ABB RAPID module: ToolPaths.mod

MODULE ToolPaths

    PERS jointtarget CurrentJoints5:=[[111.289,20.3366,35.7518,0.0387684,32.6999,-249.807],[1082.85,9E+09,9E+09,9E+09,9E+09,9E+09]];
    PERS jointtarget CurrentJoints6:=[[105.901,37.7221,15.0236,0.230043,36.0283,-255.346],[1082.85,9E+09,9E+09,9E+09,9E+09,9E+09]];


    TASK PERS wobjdata Bed1:=[FALSE,TRUE,"",[[1000.00,930.569,220.66],[1,0.000655845,-0.000507562,-0.00020191]],[[0,0,0],[1,0,0,0]]];
    !Z 185.66
    !Track -230.02 at measurement

    PERS robtarget pScreed1:=[[-1100,1500,1500],[0.00814298,0.999961,0.000966756,0.00335392],[0,-1,-2,0],[-300,9E+09,9E+09,9E+09,9E+09,9E+09]];
    PERS robtarget pScreed2:=[[-1100,1500,1500],[0.00814298,0.999961,0.000966756,0.00335392],[0,-1,-2,0],[-300,9E+09,9E+09,9E+09,9E+09,9E+09]];

    CONST num HeliOverlapMin:=450;
    CONST num PanOverlapMin:=450;
    CONST num HeliBladeWidth:=1150;
    VAR num HeliPasses;
    VAR num HeliPassWidth;
    CONST num ScreedYpos:=2955;
    CONST num wBedXmin:=1600;
    CONST num wBedXmax:=10200;
    CONST num wBedYmin:=955;
    CONST num wBedYmax:=4955;
    CONST num FormHeight:=150;
    CONST num FormWidth:=65;
    PERS num PitchZOffset:=0;

    VAR speeddata vVS:=[50,15,2000,15];
    ![mm/s TCP, degrees/s TCP, mm/s external axes, degrees/s external axes]
    VAR speeddata vHeli:=[40,10,2000,15];
    VAR speeddata vPlotter:=[1000,30,2000,15];
    VAR zonedata zVS:=z5;
    VAR zonedata zHeli:=z5;
    VAR zonedata zPlotter:=z0;


    VAR robtarget Plotterp1:=[[1000,1000,-10],[0.000337803,0.93262,-0.36086,0.000225436],[0,-1,-2,0],[3400,9E+09,9E+09,9E+09,9E+09,9E+09]];
    PERS robtarget Plotterp2:=[[-2250,790,-20],[6.12303E-17,1,0,0],[0,-1,-1,0],[8453.51,9E+09,9E+09,9E+09,9E+09,9E+09]];
    PERS robtarget Plotterp3:=[[-6000,3500,-20],[4.32964E-17,0.707107,-0.707107,-4.32964E-17],[0,-1,-1,0],[1989.63,9E+09,9E+09,9E+09,9E+09,9E+09]];
    PERS robtarget Plotterp4:=[[-6000,500,-20],[6.12303E-17,1,0,0],[1,-1,0,0],[4703.51,9E+09,9E+09,9E+09,9E+09,9E+09]];
    PERS robtarget Plotterp5:=[[1000,1000,-20],[5.65694E-17,0.92388,-0.382683,-2.34318E-17],[1,-1,0,0],[390.38,9E+09,9E+09,9E+09,9E+09,9E+09]];
    PERS robtarget Plotterc5:=[[-2250,3250,-20],[0.00237199,0.67253,-0.740066,0.000521901],[0,-1,-1,0],[0,9E+09,9E+09,9E+09,9E+09,9E+09]];
    VAR num Plotterc5r:=500;
    VAR robtarget PlotterTemp:=[[1500,3000,-10],[0.00237199,0.67253,-0.740066,0.000521901],[0,-1,-1,0],[3400,9E+09,9E+09,9E+09,9E+09,9E+09]];
    VAR robtarget PlotterTemp2:=[[1500,3000,-10],[0.00237199,0.67253,-0.740066,0.000521901],[0,-1,-1,0],[3400,9E+09,9E+09,9E+09,9E+09,9E+09]];
    VAR robtarget PlotterTemp3:=[[1500,3000,-10],[0.00237199,0.67253,-0.740066,0.000521901],[0,-1,-1,0],[3400,9E+09,9E+09,9E+09,9E+09,9E+09]];
    VAR num PlotterZ:=0;
    VAR num PlotterZOri;

    VAR robtarget pHeliStart:=[[-900,900,163.71],[0.000446787,0.711247,-0.702933,-0.00362622],[1,0,0,0],[7000,9E+09,9E+09,9E+09,9E+09,9E+09]];
    ![0.00497429,-0.71119,0.702786,0.0165738],[0,0,-1,0]
    VAR robtarget pHeliEnd:=[[-2590,2800,163.71],[0.000446787,0.711247,-0.702933,-0.00362622],[1,0,0,0],[5500,9E+09,9E+09,9E+09,9E+09,9E+09]];
    !154.71],[0.000446787,0.711247,-0.702933,-0.00362622],[1,0,0,0]
    VAR robtarget pHeliTempS;
    VAR robtarget pHeliTempE;
    VAR robtarget pHeliTemp1;
    VAR robtarget pHeliTemp2;

    VAR robtarget pScreedStart:=[[500,1900,145],[0.00523034,0.999956,0.00749019,-0.00219287],[0,-1,-2,0],[2000,9E+09,9E+09,9E+09,9E+09,9E+09]];
    VAR robtarget pScreedEnd:=[[6500,1900,145],[0.00523034,0.999956,0.00749019,-0.00219287],[0,-1,-2,0],[7700,9E+09,9E+09,9E+09,9E+09,9E+09]];


    VAR num iTaskno:=-1;
    VAR num iPlotType:=-1;
    VAR num iAngle:=-1;
    VAR num iPlotSide:=-1;
    VAR num iCoord1x:=-1;
    VAR num iCoord1y:=-1;
    VAR num iCoord2x:=-1;
    VAR num iCoord2y:=-1;
    VAR num iCoord3x:=-1;
    VAR num iCoord3y:=-1;
    VAR num iCoord4x:=-1;
    VAR num iCoord4y:=-1;
    VAR num iCoordTemp:=-1;
    VAR num iHeliBladeSpeed:=-1;
    VAR num iHeliBladeAngle:=-1;
    VAR num iZoffset:=0;
    VAR num iHeliPan:=-1;
    VAR num iLRUD:=-1;

    CONST num TieInWidth:=25;
    CONST num GroutWidth:=50;
    CONST num GroutHeight:=500;
    CONST num TriangleBase:=25;
    CONST num TriangleHeight:=50;
    CONST num PlotCircleD:=60;
    VAR num TriangleAngle:=0;
    VAR num CrossHairExt:=10;

    CONST num BedXmin:=10;
    CONST num BedXmax:=8000;
    CONST num BedYmin:=10;
    CONST num BedYmax:=3800;

    CONST num PlotA6Max:=45;
    !45;
    CONST num PlotWaitTime:=0.3;
    PERS num anglex:=179.861;
    PERS num angley:=-0.241379;
    PERS num anglez:=-95.4741;
    VAR pose Object;

    PERS num BedZread:=-8.28;

    VAR robtarget p10maps:=[[-350,150,250],[0.00321343,0.67631,-0.736609,0.000689698],[0,0,-1,0],[7700,9E+09,9E+09,9E+09,9E+09,9E+09]];

    !VAR num BedZreads{4,24}:=[
    !  [13.28, 12.88, 12.68, 14.03, 15.46, 10.94,  8.17,  6.79,  4.83,  2.37,  0.97,  0.30,  0.00,  0.24,  0.47, 0, 0, 0, 0, 0, 0, 0, 0, 0],
    !  [15.76, 14.97, 14.36, 15.69, 16.55, 13.22, 10.94,  9.86,  7.97,  6.00,  4.27,  3.57,  2.82,  2.70,  1.69, 0, 0, 0, 0, 0, 0, 0, 0, 0],
    !  [16.92, 16.33, 16.18, 17.01, 17.20, 14.79, 12.97, 12.12, 10.27,  8.39,  6.92,  5.72,  4.82,  4.65,  2.84, 0, 0, 0, 0, 0, 0, 0, 0, 0],
    !  [17.97, 18.08, 18.34, 18.15, 17.16, 15.42, 14.97, 14.02, 12.65, 11.42,  9.54,  8.23,  6.97,  6.59,  4.58, 0, 0, 0, 0, 0, 0, 0, 0, 0]
    !];

    VAR num BedZreads{4,24}:=[
  [2.28,1.88,1.68,3.03,4.46,-0.06,-2.83,-4.21,-6.17,-8.63,-10.03,-10.70,-11.00,-10.76,-10.53,0,0,0,0,0,0,0,0,0],
  [4.76,3.97,3.36,4.69,5.55,2.22,-0.06,-1.14,-3.03,-5.00,-6.73,-7.43,-8.18,-8.30,-9.31,0,0,0,0,0,0,0,0,0],
  [5.92,5.33,5.18,6.01,6.20,3.79,1.97,1.12,-0.73,-2.61,-4.08,-5.28,-6.18,-6.35,-8.16,0,0,0,0,0,0,0,0,0],
  [6.97,7.08,7.34,7.15,6.16,4.42,3.97,3.02,1.65,0.42,-1.46,-2.77,-4.03,-4.41,-6.42,0,0,0,0,0,0,0,0,0]
];

    VAR num BedZpos{4,24,2}:=[[
    [-350,2100],[-850,2100],[-1350,2100],[-1850,2100],[-2350,2100],[-2850,2100],[-3350,2100],[-3850,2100],[-4350,2100],[-4850,2100],[-5350,2100],[-5850,2100],[-6350,2100],[-6850,2100],[-7350,2100],[-7850,2100],[-8350,2100],[0,0],[0,0],[0,0],[0,0],[0,0],[0,0],[0,0]],

   [[-350,1450],[-850,1450],[-1350,1450],[-1850,1450],[-2350,1450],[-2850,1450],[-3350,1450],[-3850,1450],[-4350,1450],[-4850,1450],[-5350,1450],[-5850,1450],[-6350,1450],[-6850,1450],[-7350,1450],[-7850,1450],[-8350,1450],[0,0],[0,0],[0,0],[0,0],[0,0],[0,0],[0,0]],

   [[-350,800],[-850,800],[-1350,800],[-1850,800],[-2350,800],[-2850,800],[-3350,800],[-3850,800],[-4350,800],[-4850,800],[-5350,800],[-5850,800],[-6350,800],[-6850,800],[-7350,800],[-7850,800],[-8350,800],[0,0],[0,0],[0,0],[0,0],[0,0],[0,0],[0,0]],

    [[-350,150],[-850,150],[-1350,150],[-1850,150],[-2350,150],[-2850,150],[-3350,150],[-3850,150],[-4350,150],[-4850,150],[-5350,150],[-5850,150],[-6350,150],[-6850,150],[-7350,150],[-7850,150],[-8350,150],[0,0],[0,0],[0,0],[0,0],[0,0],[0,0],[0,0]]];


    PERS num Bed1Zread{10,20}:=[[0,0,0,0,0,0,0,0,0,0,0,0,0,0,0,0,0,0,0,0],
                                 [0,0,0,0,0,0,0,0,0,0,0,0,0,0,0,0,0,0,0,0],
                                 [0,0,0,0,0,0,0,0,0,0,0,0,0,0,0,0,0,0,0,0],
                                 [0,0,0,0,0,0,0,0,0,0,0,0,0,0,0,0,0,0,0,0],
                                 [0,0,0,0,0,0,0,0,0,0,0,0,0,0,0,0,0,0,0,0],
                                 [0,0,0,0,0,0,0,0,0,0,0,0,0,0,0,0,0,0,0,0],
                                 [0,0,0,0,0,0,0,0,0,0,0,0,0,0,0,0,0,0,0,0],
                                 [0,0,0,0,0,0,0,0,0,0,0,0,0,0,0,0,0,0,0,0],
                                 [0,0,0,0,0,0,0,0,0,0,0,0,0,0,0,0,0,0,0,0],
                                 [0,0,0,0,0,0,0,0,0,0,0,0,0,0,0,0,0,0,0,0]];

    PERS num Bed1Zpos{10,20,2}:=[[[0,0],[0,0],[0,0],[0,0],[0,0],[0,0],[0,0],[0,0],[0,0],[0,0],[0,0],[0,0],[0,0],[0,0],[0,0],[0,0],[0,0],[0,0],[0,0],[0,0]],

                               [[0,0],[0,0],[0,0],[0,0],[0,0],[0,0],[0,0],[0,0],[0,0],[0,0],[0,0],[0,0],[0,0],[0,0],[0,0],[0,0],[0,0],[0,0],[0,0],[0,0]],

                               [[0,0],[0,0],[0,0],[0,0],[0,0],[0,0],[0,0],[0,0],[0,0],[0,0],[0,0],[0,0],[0,0],[0,0],[0,0],[0,0],[0,0],[0,0],[0,0],[0,0]],

                               [[0,0],[0,0],[0,0],[0,0],[0,0],[0,0],[0,0],[0,0],[0,0],[0,0],[0,0],[0,0],[0,0],[0,0],[0,0],[0,0],[0,0],[0,0],[0,0],[0,0]],

                               [[0,0],[0,0],[0,0],[0,0],[0,0],[0,0],[0,0],[0,0],[0,0],[0,0],[0,0],[0,0],[0,0],[0,0],[0,0],[0,0],[0,0],[0,0],[0,0],[0,0]],

                               [[0,0],[0,0],[0,0],[0,0],[0,0],[0,0],[0,0],[0,0],[0,0],[0,0],[0,0],[0,0],[0,0],[0,0],[0,0],[0,0],[0,0],[0,0],[0,0],[0,0]],

                               [[0,0],[0,0],[0,0],[0,0],[0,0],[0,0],[0,0],[0,0],[0,0],[0,0],[0,0],[0,0],[0,0],[0,0],[0,0],[0,0],[0,0],[0,0],[0,0],[0,0]],

                               [[0,0],[0,0],[0,0],[0,0],[0,0],[0,0],[0,0],[0,0],[0,0],[0,0],[0,0],[0,0],[0,0],[0,0],[0,0],[0,0],[0,0],[0,0],[0,0],[0,0]],

                               [[0,0],[0,0],[0,0],[0,0],[0,0],[0,0],[0,0],[0,0],[0,0],[0,0],[0,0],[0,0],[0,0],[0,0],[0,0],[0,0],[0,0],[0,0],[0,0],[0,0]],

                               [[0,0],[0,0],[0,0],[0,0],[0,0],[0,0],[0,0],[0,0],[0,0],[0,0],[0,0],[0,0],[0,0],[0,0],[0,0],[0,0],[0,0],[0,0],[0,0],[0,0]]];

    CONST num XGridSpacing:=460;
    CONST num YGridSpacing:=400;


    PERS num ScrInitialD:=50;

    PERS num HeliZOffs:=0;
    !Offset based on bed heights

    VAR num SEnddiv:=0;
    VAR num SStartdiv:=0;

    VAR num ScrBedZ;

    PERS num HeliZArray{30}:=[-50,-50,-50,-50,-50,-50,-50,-50,-50,-50,-50,-50,-50,-50,-50,-50,-50,-50,-50,-50,-50,-50,-50,-50,-50,-50,-50,-50,-50,-50];
    VAR bool WithinBlades:=FALSE;
    PERS num HeliZArrayCounter:=1;
    PERS num HeliDiv:=12;
    PERS num PreviousHighest:=-50;

    !CONST robtarget p10:=[[-8200.58,3455.68,-35.54],[0.000477585,0.709995,-0.70418,0.00603077],[1,-1,0,0],[700.099,9E+09,9E+09,9E+09,9E+09,9E+09]];
    CONST robtarget pVacStart:=[[-8200.58,3455.68,-35.54],[0.00615322,-0.709926,0.704246,-0.00239206],[1,-1,0,0],[700,9E+09,9E+09,9E+09,9E+09,9E+09]];
    CONST robtarget pVacStart2:=[[-72.58,1432.35,-35.54],[0.00615322,-0.709926,0.704246,-0.00239206],[1,-1,0,0],[8680,9E+09,9E+09,9E+09,9E+09,9E+09]];
    VAR num iTask:=-1;
    VAR num iPete:=-1;
    VAR num PeteXoffset:=0;
    VAR num PeteYoffset:=0;
    VAR num FormStartX:=7300;
    VAR num FormStartY:=3500;
    VAR num FormXLength:=4750;
    VAR num FormYlength:=1800;
    VAR num CrnrMarkLngth:=300;
    VAR speeddata PanTrvSpd:=[100,30,2000,15];
    VAR num PanBldSpd:=70;
    VAR num PanZOffset:=0;
    VAR num VSZOffset:=0;
    VAR num VSAngleOffset:=0;
    VAR num DummyRun:=0;
    VAR num DummyZOffs:=0;

    PROC PetePanels()
        PeteYoffset:=0;
        PeteXoffset:=0;
        TPErase;
        TPReadNum iTask,"1:Home,2:PackAway,3:Sync,4:Py_28-jan_4:34pm";
        TEST iTask
        CASE 1:
            Home;
        CASE 4:
            FormXLength:=4750;
            FormYlength:=1800;
            TPErase;
            TPWrite "8:Datum,9:PyHeli,10:PyVac,11:PyPolish";
            TPWrite "12:PyVibScreed,13:PyPan";
            TPReadNum iTaskno,"Enter task #:";
            TEST iTaskno
            CASE 1:
                !                TPReadNum iPete,"Enter X  offset (+mm moves closer to the tools)";
                !                IF iPete>(FormStartX-FormXLength-300) OR iPete<0 THEN
                !                    TPWrite "Invalid offset";
                !                    Stop;
                !                    EXIT;
                !                ELSE
                !                    PeteXoffset:=iPete;
                !                ENDIF

                !                TPReadNum iPete,"Enter Y  offset (+mm moves closer to the track)";
                !                IF iPete>(FormStartY-FormYLength-300) OR iPete<0 THEN
                !                    TPWrite "Invalid offset";
                !                    Stop;
                !                    EXIT;
                !                ELSE
                !                    PeteYoffset:=iPete;
                !                ENDIF

                !Formbox
                PlotRect(FormStartX-FormXLength-PeteXoffset-FormWidth),(FormStartY-FormYLength-PeteYoffset-FormWidth),(FormStartX-FormXLength-PeteXoffset-FormWidth),(FormStartY-PeteYoffset+FormWidth),(FormStartX-PeteXoffset+FormWidth),(FormStartY-PeteYoffset+FormWidth),(FormStartX-PeteXoffset+FormWidth),(FormStartY-FormYLength-PeteYoffset-FormWidth);
                CurrentJoints:=CJointT();
                CurrentPos:=CalcRobT(CurrentJoints,tPlotter\WObj:=Bed1Wyong);
                MoveL Offs(CurrentPos,0,0,(1000-CurrentPos.trans.z)),v100,z5,tPlotter\WObj:=Bed1Wyong;

                PlotlineStartLift(FormStartX-FormXLength-PeteXoffset+CrnrMarkLngth),(FormStartY-FormYLength-PeteYoffset),(FormStartX-FormXLength-PeteXoffset),(FormStartY-FormYLength-PeteYoffset);
                PlotLineEndLift(FormStartX-FormXLength-PeteXoffset),(FormStartY-FormYLength-PeteYoffset),(FormStartX-FormXLength-PeteXoffset),(FormStartY-FormYLength-PeteYoffset-CrnrMarkLngth);

                PlotlineStartLift(FormStartX-FormXLength-PeteXoffset),(FormStartY-PeteYoffset-CrnrMarkLngth),(FormStartX-FormXLength-PeteXoffset),(FormStartY-PeteYoffset);
                PlotLineEndLift(FormStartX-FormXLength-PeteXoffset),(FormStartY-PeteYoffset),(FormStartX-FormXLength-PeteXoffset+CrnrMarkLngth),(FormStartY-PeteYoffset);


                !Ferrules
                iCoord1x:=FormStartX-600-PeteXoffset;
                iCoord1y:=FormStartY-1480-PeteYoffset;
                PlotCirc iCoord1x,iCoord1y,(PlotCircleD/2);
                PlotLine(iCoord1x-PlotCircleD/2-CrossHairExt),iCoord1y,(iCoord1x+PlotCircleD/2+CrossHairExt),iCoord1y;
                PlotLine iCoord1x,(iCoord1y-PlotCircleD/2-CrossHairExt),iCoord1x,(iCoord1y+PlotCircleD/2+CrossHairExt);
                !Lifters
                iCoord1x:=FormStartX-FormXLength-PeteXoffset;
                iCoord1y:=FormStartY+620-FormYlength-PeteYoffset;
                TriangleAngle:=0;
                PlotLineStartLift iCoord1x-TriangleBase/2*Sin(TriangleAngle),iCoord1y-TriangleBase/2*Cos(TriangleAngle),iCoord1x+TriangleBase/2*Sin(TriangleAngle),iCoord1y+TriangleBase/2*Cos(TriangleAngle);
                PlotLineNoLift iCoord1x+TriangleBase/2*Sin(TriangleAngle),iCoord1y+TriangleBase/2*Cos(TriangleAngle),iCoord1x+TriangleHeight*Cos(TriangleAngle),iCoord1y-TriangleHeight*Sin(TriangleAngle);
                PlotLineEndLift iCoord1x+TriangleHeight*Cos(TriangleAngle),iCoord1y-TriangleHeight*Sin(TriangleAngle),iCoord1x-TriangleBase/2*Sin(TriangleAngle),iCoord1y-TriangleBase/2*Cos(TriangleAngle);

                iCoord1x:=FormStartX-FormXLength-PeteXoffset;
                iCoord1y:=FormStartY-620-PeteYoffset;
                TriangleAngle:=0;
                PlotLineStartLift iCoord1x-TriangleBase/2*Sin(TriangleAngle),iCoord1y-TriangleBase/2*Cos(TriangleAngle),iCoord1x+TriangleBase/2*Sin(TriangleAngle),iCoord1y+TriangleBase/2*Cos(TriangleAngle);
                PlotLineNoLift iCoord1x+TriangleBase/2*Sin(TriangleAngle),iCoord1y+TriangleBase/2*Cos(TriangleAngle),iCoord1x+TriangleHeight*Cos(TriangleAngle),iCoord1y-TriangleHeight*Sin(TriangleAngle);
                PlotLineEndLift iCoord1x+TriangleHeight*Cos(TriangleAngle),iCoord1y-TriangleHeight*Sin(TriangleAngle),iCoord1x-TriangleBase/2*Sin(TriangleAngle),iCoord1y-TriangleBase/2*Cos(TriangleAngle);

                iCoord1x:=FormStartX+350-FormXLength-PeteXoffset;
                iCoord1y:=FormStartY-PeteYoffset;
                TriangleAngle:=0;
                PlotLineStartLift iCoord1x-TriangleHeight*Sin(TriangleAngle),iCoord1y-TriangleHeight*Cos(TriangleAngle),iCoord1x-TriangleBase/2*Cos(TriangleAngle),iCoord1y+TriangleBase/2*Sin(TriangleAngle);
                PlotLineNoLift iCoord1x-TriangleBase/2*Cos(TriangleAngle),iCoord1y+TriangleBase/2*Sin(TriangleAngle),iCoord1x+TriangleBase/2*Cos(TriangleAngle),iCoord1y-TriangleBase/2*Sin(TriangleAngle);
                PlotLineEndLift iCoord1x+TriangleBase/2*Cos(TriangleAngle),iCoord1y-TriangleBase/2*Sin(TriangleAngle),iCoord1x-TriangleHeight*Sin(TriangleAngle),iCoord1y-TriangleHeight*Cos(TriangleAngle);

                iCoord1x:=FormStartX+2170-FormXLength-PeteXoffset;
                iCoord1y:=FormStartY-PeteYoffset;
                TriangleAngle:=0;
                PlotLineStartLift iCoord1x-TriangleHeight*Sin(TriangleAngle),iCoord1y-TriangleHeight*Cos(TriangleAngle),iCoord1x-TriangleBase/2*Cos(TriangleAngle),iCoord1y+TriangleBase/2*Sin(TriangleAngle);
                PlotLineNoLift iCoord1x-TriangleBase/2*Cos(TriangleAngle),iCoord1y+TriangleBase/2*Sin(TriangleAngle),iCoord1x+TriangleBase/2*Cos(TriangleAngle),iCoord1y-TriangleBase/2*Sin(TriangleAngle);
                PlotLineEndLift iCoord1x+TriangleBase/2*Cos(TriangleAngle),iCoord1y-TriangleBase/2*Sin(TriangleAngle),iCoord1x-TriangleHeight*Sin(TriangleAngle),iCoord1y-TriangleHeight*Cos(TriangleAngle);

                iCoord1x:=FormStartX-2170-PeteXoffset;
                iCoord1y:=FormStartY-PeteYoffset;
                TriangleAngle:=0;
                PlotLineStartLift iCoord1x-TriangleHeight*Sin(TriangleAngle),iCoord1y-TriangleHeight*Cos(TriangleAngle),iCoord1x-TriangleBase/2*Cos(TriangleAngle),iCoord1y+TriangleBase/2*Sin(TriangleAngle);
                PlotLineNoLift iCoord1x-TriangleBase/2*Cos(TriangleAngle),iCoord1y+TriangleBase/2*Sin(TriangleAngle),iCoord1x+TriangleBase/2*Cos(TriangleAngle),iCoord1y-TriangleBase/2*Sin(TriangleAngle);
                PlotLineEndLift iCoord1x+TriangleBase/2*Cos(TriangleAngle),iCoord1y-TriangleBase/2*Sin(TriangleAngle),iCoord1x-TriangleHeight*Sin(TriangleAngle),iCoord1y-TriangleHeight*Cos(TriangleAngle);

                iCoord1x:=FormStartX-350-PeteXoffset;
                iCoord1y:=FormStartY-PeteYoffset;
                TriangleAngle:=0;
                PlotLineStartLift iCoord1x-TriangleHeight*Sin(TriangleAngle),iCoord1y-TriangleHeight*Cos(TriangleAngle),iCoord1x-TriangleBase/2*Cos(TriangleAngle),iCoord1y+TriangleBase/2*Sin(TriangleAngle);
                PlotLineNoLift iCoord1x-TriangleBase/2*Cos(TriangleAngle),iCoord1y+TriangleBase/2*Sin(TriangleAngle),iCoord1x+TriangleBase/2*Cos(TriangleAngle),iCoord1y-TriangleBase/2*Sin(TriangleAngle);
                PlotLineEndLift iCoord1x+TriangleBase/2*Cos(TriangleAngle),iCoord1y-TriangleBase/2*Sin(TriangleAngle),iCoord1x-TriangleHeight*Sin(TriangleAngle),iCoord1y-TriangleHeight*Cos(TriangleAngle);

                PlotlineStartLift(FormStartX-PeteXoffset-CrnrMarkLngth),(FormStartY-PeteYoffset),(FormStartX-PeteXoffset+FormWidth),(FormStartY-PeteYoffset+FormWidth);
                PlotLineEndLift(FormStartX-PeteXoffset+FormWidth),(FormStartY-PeteYoffset+FormWidth),(FormStartX-PeteXoffset+FormWidth),(FormStartY-PeteYoffset+FormWidth-CrnrMarkLngth);

                !Grout tubes
                iCoord1x:=FormStartX-PeteXoffset;
                iCoord1y:=FormStartY-150-PeteYoffset;
                PlotLine iCoord1x,iCoord1y,(iCoord1x-350),iCoord1y;
                PlotCirc(iCoord1x-300),icoord1y,(PlotCircleD/2);

                iCoord1x:=FormStartX-PeteXoffset;
                iCoord1y:=FormStartY+150-FormYlength-PeteYoffset;
                PlotLine iCoord1x,iCoord1y,(iCoord1x-350),iCoord1y;
                PlotCirc(iCoord1x-300),icoord1y,(PlotCircleD/2);

                PlotlineStartLift(FormStartX-PeteXoffset),(FormStartY-FormYLength-PeteYoffset+CrnrMarkLngth),(FormStartX-PeteXoffset),(FormStartY-FormYLength-PeteYoffset);
                PlotLineEndLift(FormStartX-PeteXoffset),(FormStartY-FormYLength-PeteYoffset),(FormStartX-PeteXoffset-CrnrMarkLngth),(FormStartY-FormYLength-PeteYoffset);

                CurrentJoints:=CJointT();
                CurrentPos:=CalcRobT(CurrentJoints,tPlotter\WObj:=Bed1Wyong);
                MoveL Offs(CurrentPos,0,0,(1000-CurrentPos.trans.z)),v100,z5,tPlotter\WObj:=Bed1Wyong;

                Home;
            CASE 2:
                !                TPReadNum iPete,"Enter X  offset (+mm moves closer to the tools)";
                !                IF iPete>(FormStartX-FormXLength-300) OR iPete<0 THEN
                !                    TPWrite "Invalid offset";
                !                    Stop;
                !                    EXIT;
                !                ELSE
                !                    PeteXoffset:=iPete;
                !                ENDIF

                !                TPReadNum iPete,"Enter Y  offset (+mm moves closer to the track)";
                !                IF iPete>(FormStartY-FormYLength-300) OR iPete<0 THEN
                !                    TPWrite "Invalid offset";
                !                    Stop;
                !                    EXIT;
                !                ELSE
                !                    PeteYoffset:=iPete;
                !                ENDIF
                TPReadNum iPete,"Enter angle offset (+deg angles front down)";
                IF iPete>15 OR iPete<-15 THEN
                    TPWrite "Invalid angle offset";
                    Stop;
                    EXIT;
                ELSE
                    VSAngleOffset:=iPete;
                ENDIF

                TPReadNum iPete,"Enter Z offset(+mm{400max} moves higher, -mm pushes down more)";
                IF iPete>400 OR iPete<-50 THEN
                    TPWrite "Invalid Z offset";
                    Stop;
                    EXIT;
                ELSE
                    VSZOffset:=iPete;
                ENDIF

                Screed(FormStartX-FormXLength-PeteXoffset),(FormStartX-PeteXoffset),VSZOffset,VSAngleOffset;
                Home;
            CASE 3:
                Polish;
                Home;
            CASE 4:
                VacuumBed;
                Home;
            CASE 5:

                TPReadNum iPete,"Enter 0 real run, 1 for dummmy run";
                IF iPete<>0 AND iPete<>1 THEN
                    TPWrite "Invalid entry";
                    Stop;
                    EXIT;
                ELSE
                    DummyRun:=iPete;
                ENDIF

                TPReadNum iPete,"Enter Y offset (+mm moves further away from track)";
                IF iPete>FormYLength OR iPete<0 THEN
                    TPWrite "Invalid offset";
                    Stop;
                    EXIT;
                ELSE
                    FCHeliOffs:=iPete;
                    FCHeliStartX:=FormStartX-FormXLength;
                    FCHeliStartY:=FormStartY-FormYlength+FCHeliOffs;
                    FCHeliEndX:=FormStartX;
                ENDIF

                TPReadNum iPete,"Enter Heli travel speed, mm/s(options: 5,10,20,30,40,50,60,80,100,150,200,500)";
                IF iPete=5 OR iPete=10 OR iPete=20 OR iPete=30 OR iPete=40 OR iPete=50 OR iPete=60 OR iPete=80 OR iPete=100 OR iPete=150 OR iPete=200 OR iPete=500 THEN
                    FCHeliSpd.v_tcp:=iPete;
                ELSE
                    TPWrite "Invalid travel speed";
                    Stop;
                    EXIT;
                ENDIF

                IF DummyRun=0 THEN

                    TPReadNum iPete,"Enter Heli blade speed (either 70, 100 or 140 rpm)";
                    FCHeliBldSpd:=iPete;
                    IF iPete=140 THEN
                        FCHeliLD:=HeliLoad140rpm;
                    ELSEIF iPete=100 THEN
                        FCHeliLD:=HeliLoad100rpm;
                    ELSEIF iPete=70 THEN
                        FCHeliLD:=HeliLoad70rpm;
                    ELSE
                        TPWrite "Invalid blade speed";
                        Stop;
                        EXIT;
                    ENDIF

                    TPReadNum iPete,"Enter blade angle (0 to 10 degrees)";
                    IF iPete>10 OR iPete<0 THEN
                        TPWrite "Invalid blade angle";
                        Stop;
                        EXIT;
                    ELSE
                        FCBladeAngle:=iPete;
                    ENDIF

                    TPReadNum iPete,"Enter Force in Newtons (robot will press down with this value, 1300 max)";
                    IF iPete>1300 OR iPete<0 THEN
                        TPWrite "Invalid offset";
                        Stop;
                        EXIT;
                    ELSE
                        FCHeliFrce:=iPete;
                    ENDIF

                    HeliFC FCHeliStartX,FCHeliStartY,FCHeliEndX,FCHeliSpd,FCHeliBldSpd,FCBladeAngle,FCHeliFrce,FCHeliLD;
                ELSEIF DummyRun=1 THEN
                    HeliFCDummy FCHeliStartX,FCHeliStartY,FCHeliEndX,FCHeliSpd;
                ELSE
                    TPWrite "Invalid selection";
                    Stop;
                    EXIT;
                ENDIF

            CASE 6:

                TPReadNum iPete,"Enter Pan travel speed, mm/s(options: 5,10,20,30,40,50,60,80,100,150,200,500)";
                IF iPete=5 OR iPete=10 OR iPete=20 OR iPete=30 OR iPete=40 OR iPete=50 OR iPete=60 OR iPete=80 OR iPete=100 OR iPete=150 OR iPete=200 OR iPete=500 THEN
                    PanTrvSpd.v_tcp:=iPete;
                ELSE
                    TPWrite "Invalid travel speed";
                    Stop;
                    EXIT;
                ENDIF

                TPReadNum iPete,"Enter 0 real run, 1 for dummmy run";
                IF iPete<>0 AND iPete<>1 THEN
                    TPWrite "Invalid entry";
                    Stop;
                    EXIT;
                ELSE
                    DummyRun:=iPete;
                ENDIF

                IF DummyRun=0 THEN

                    TPReadNum iPete,"Pan rotation speed (rpm, 40-140)";
                    IF iPete>140 OR iPete<40 THEN
                        TPWrite "Invalid Heli speed.";
                        Stop;
                        EXIT;
                    ELSE
                        PanBldSpd:=iPete;
                    ENDIF

                    TPReadNum iPete,"Enter Z offset (+mm has heli higher, -mm pushes down more)";
                    IF iPete>400 OR iPete<-50 THEN
                        TPWrite "Invalid offset";
                        Stop;
                        EXIT;
                    ELSE
                        PanZOffset:=iPete;
                    ENDIF

                    HeliPanLR(FormStartX-FormXLength-PeteXoffset),(FormStartY-FormYLength-PeteYoffset),(FormStartX-PeteXoffset),2500,PanTrvSpd,PanBldSpd,PanZOffset;
                ELSE
                    TPWrite "Invalid selection";
                    Stop;
                    EXIT;
                ENDIF


            CASE 7:
                PolishTest;
            CASE 8:
                Datum;
            CASE 9:
                PyHeli;
            CASE 10:
                PyVac;
            CASE 11:
                PyPolish;
            CASE 12:
                PyVibScreed;
            CASE 13:
                PyPan;
            DEFAULT:
                RAISE ERR_INVALID_INPUT;
            ENDTEST

        CASE 2:
            PackAway;
        CASE 3:
            MoveAbsJ [[86.92,9.65,27.89,0.50,50.60,-4.00],[1388.98,9E9,9E9,9E9,9E9,9E9]],v100,fine,tool0;
            Stop;
        DEFAULT:
            RAISE ERR_INVALID_INPUT;
        ENDTEST
    ERROR
        RAISE ;
    ENDPROC


    PROC DemoScreen()
        TPErase;
        TPReadNum iTask,"1: Demo, 2: Production";
        TEST iTask
        CASE 1:
            TPErase;
            TPReadNum iTaskno,"Enter Demo #: 1: Home, 2: Plot 3: Screed, 4: Polish, 5: Vac";
            TEST iTaskno
            CASE 1:
                Home;
            CASE 2:
                RobbiePlot;
            CASE 3:
                Screed 500,6000,0,11;
            CASE 4:
                PolishDemo;
            CASE 5:
                VacuumBed;
            DEFAULT:
                RAISE ERR_INVALID_INPUT;
            ENDTEST

        CASE 2:
            TaskToDo;
        DEFAULT:
            RAISE ERR_INVALID_INPUT;
        ENDTEST
    ERROR
        RAISE ;
    ENDPROC


    PROC TaskToDo()
        TPErase;
        TPReadNum iTaskno,"Enter task #: 1: Home, 2: Loadout 3: Plot, 4: Screed, 5: Heli, 6: Vac, 7: Polish";
        TEST iTaskno
        CASE 1:
            Home;
        CASE 2:
            Home;
            MoveJ pHomeLoadout,v500,z50,tTCMaster;
        CASE 3:
            TPErase;
            TPWrite "Plotting: Enter 1 for formbox, 2 for circle/cross, 3 for grout tube,";
            TPWrite " 4 for square/cross, 5 for triangle.";
            TPReadNum iPlotType,"Enter Selection:";
            TPErase;
            IF iPlotType=1 THEN
                !Form box
                TPWrite "Enter the coordinates for each corner of the formwork.";
                TPReadNum iCoord1x,"Enter first coordinate X value";
                TPReadNum iCoord1y,"Enter first coordinate y value";
                TPReadNum iCoord2x,"Enter second coordinate X value";
                TPReadNum iCoord2y,"Enter second coordinate y value";
                TPReadNum iCoord3x,"Enter third coordinate X value";
                TPReadNum iCoord3y,"Enter third coordinate y value";
                TPReadNum iCoord4x,"Enter fourth coordinate X value";
                TPReadNum iCoord4y,"Enter fourth coordinate y value";
                IF iCoord1x<BedXmin OR iCoord1y<BedYmin OR iCoord2x<BedXmin OR iCoord2y<BedYmin OR iCoord3x<BedXmin OR iCoord3y<BedYmin OR iCoord4x<BedXmin OR iCoord4y<BedYmin OR iCoord1x>BedXmax OR iCoord1y>BedYmax OR iCoord2x>BedXmax OR iCoord2y>BedYmax OR iCoord3x>BedXmax OR iCoord3y>BedYmax OR iCoord4x>BedXmax OR iCoord4y>BedYmax OR (iCoord1x*iCoord1x+iCoord1y*iCoord1y<2560000) OR (iCoord2x*iCoord2x+iCoord2y*iCoord2y<2560000) OR (iCoord3x*iCoord3x+iCoord3y*iCoord3y<2560000) OR (iCoord4x*iCoord4x+iCoord4y*iCoord4y<2560000) THEN
                    RAISE ERR_INVALID_INPUT;
                ENDIF
                PlotRect iCoord1x,iCoord1y,iCoord2x,iCoord2y,iCoord3x,iCoord3y,iCoord4x,iCoord4y;

            ELSEIF iPlotType=2 THEN
                !ferrule - Circle with cross
                TPWrite "Enter the coordinates for the centre position of the ferrule.";
                TPReadNum iCoord1x,"Enter centre coordinate X value";
                TPReadNum iCoord1y,"Enter centre coordinate y value";

                IF (iCoord1x-PlotCircleD)<BedXmin OR (iCoord1y-PlotCircleD)<BedYmin OR (iCoord1x+PlotCircleD)>BedXmax OR (iCoord1y+PlotCircleD)>BedYmax OR ((iCoord1x-PlotCircleD)*(iCoord1x-PlotCircleD)+(iCoord1y-PlotCircleD)*(iCoord1y-PlotCircleD)<2560000) THEN
                    RAISE ERR_INVALID_INPUT;
                ENDIF
                PlotCirc iCoord1x,iCoord1y,(PlotCircleD/2);
                PlotLine(iCoord1x-PlotCircleD/2-CrossHairExt),iCoord1y,(iCoord1x+PlotCircleD/2+CrossHairExt),iCoord1y;
                PlotLine iCoord1x,(iCoord1y-PlotCircleD/2-CrossHairExt),iCoord1x,(iCoord1y+PlotCircleD/2+CrossHairExt);

            ELSEIF iPlotType=3 THEN
                !Grout Rectangle
                TPWrite "Enter the edge coordinate coordinate, followed by the angle.";
                TPReadNum iCoord1x,"Enter centre coordinate X value";
                TPReadNum iCoord1y,"Enter centre coordinate y value";
                TPWrite "0 degrees is perpendicular, -90 degrees is left/CCW, +90 is right/CW.,";
                TPReadNum iAngle,"Enter the angle";
                TPErase;
                TPWrite "Enter the side for the grout tube to be placed.";
                TPWrite " ------3------ ";
                TPWrite " |           | ";
                TPWrite "2|     X     |4";
                TPWrite " |           | ";
                TPWrite " ------1------ ";
                TPWrite "ROBOT/TRACK SIDE";
                TPReadNum iPlotSide,"Enter side:";

                IF iAngle<-90 OR iAngle>90 THEN
                    RAISE ERR_INVALID_INPUT;
                ENDIF

                TEST iPlotSide
                CASE 1:
                    IF iCoord1x-GroutWidth/2*Cos(iAngle)<BedXmin OR iCoord1y+GroutWidth/2*Sin(iAngle)<BedYmin OR iCoord1x-GroutWidth/2*Cos(iAngle)+GroutHeight*Sin(iAngle)<BedXmin OR iCoord1y+GroutHeight*Cos(iAngle)+GroutWidth/2*Sin(iAngle)<BedYmin OR iCoord1x+GroutWidth/2*Cos(iAngle)+GroutHeight*Sin(iAngle)<BedXmin OR iCoord1y+GroutHeight*Cos(iAngle)-GroutWidth/2*Sin(iAngle)<BedYmin OR iCoord1x+GroutWidth/2*Cos(iAngle)<BedXmin OR iCoord1y-GroutWidth/2*Sin(iAngle)<BedYmin OR ((iCoord1x-GroutHeight)*(iCoord1x-GroutWidth)+(iCoord1y-GroutHeight)*(iCoord1y-GroutWidth)<2560000) THEN
                        RAISE ERR_INVALID_INPUT;
                    ENDIF

                    IF iCoord1x-GroutWidth/2*Cos(iAngle)>BedXmax OR iCoord1y+GroutWidth/2*Sin(iAngle)>BedYmax OR iCoord1x-GroutWidth/2*Cos(iAngle)+GroutHeight*Sin(iAngle)>BedXmax OR iCoord1y+GroutHeight*Cos(iAngle)+GroutWidth/2*Sin(iAngle)>BedYmax OR iCoord1x+GroutWidth/2*Cos(iAngle)+GroutHeight*Sin(iAngle)>BedXmax OR iCoord1y+GroutHeight*Cos(iAngle)-GroutWidth/2*Sin(iAngle)>BedYmax OR iCoord1x+GroutWidth/2*Cos(iAngle)>BedXmax OR iCoord1y-GroutWidth/2*Sin(iAngle)>BedYmax THEN
                        RAISE ERR_INVALID_INPUT;
                    ENDIF

                    PlotRect iCoord1x-GroutWidth/2*Cos(iAngle),iCoord1y+GroutWidth/2*Sin(iAngle),iCoord1x-GroutWidth/2*Cos(iAngle)+GroutHeight*Sin(iAngle),iCoord1y+GroutHeight*Cos(iAngle)+GroutWidth/2*Sin(iAngle),iCoord1x+GroutWidth/2*Cos(iAngle)+GroutHeight*Sin(iAngle),iCoord1y+GroutHeight*Cos(iAngle)-GroutWidth/2*Sin(iAngle),iCoord1x+GroutWidth/2*Cos(iAngle),iCoord1y-GroutWidth/2*Sin(iAngle);

                CASE 2:

                    IF iCoord1x-GroutWidth/2*Sin(iAngle)<BedXmin OR iCoord1y-GroutWidth/2*Cos(iAngle)<BedYmin OR iCoord1x+GroutWidth/2*Sin(iAngle)<BedXmin OR iCoord1y+GroutWidth/2*Cos(iAngle)<BedYmin OR iCoord1x+GroutWidth/2*Sin(iAngle)+GroutHeight*Cos(iAngle)<BedXmin OR iCoord1y-GroutHeight*Sin(iAngle)+GroutWidth/2*Cos(iAngle)<BedYmin OR iCoord1x-GroutWidth/2*Sin(iAngle)+GroutHeight*Cos(iAngle)<BedXmin OR iCoord1y-GroutHeight*Sin(iAngle)-GroutWidth/2*Cos(iAngle)<BedYmin OR ((iCoord1x-GroutHeight)*(iCoord1x-GroutWidth)+(iCoord1y-GroutHeight)*(iCoord1y-GroutWidth)<2560000) THEN
                        RAISE ERR_INVALID_INPUT;
                    ENDIF

                    IF iCoord1x-GroutWidth/2*Sin(iAngle)>BedXmax OR iCoord1y-GroutWidth/2*Cos(iAngle)>BedYmax OR iCoord1x+GroutWidth/2*Sin(iAngle)>BedXmax OR iCoord1y+GroutWidth/2*Cos(iAngle)>BedYmax OR iCoord1x+GroutWidth/2*Sin(iAngle)+GroutHeight*Cos(iAngle)>BedXmax OR iCoord1y-GroutHeight*Sin(iAngle)+GroutWidth/2*Cos(iAngle)>BedYmax OR iCoord1x-GroutWidth/2*Sin(iAngle)+GroutHeight*Cos(iAngle)>BedXmax OR iCoord1y-GroutHeight*Sin(iAngle)-GroutWidth/2*Cos(iAngle)>BedYmax THEN
                        RAISE ERR_INVALID_INPUT;
                    ENDIF

                    PlotRect iCoord1x-GroutWidth/2*Sin(iAngle),iCoord1y-GroutWidth/2*Cos(iAngle),iCoord1x+GroutWidth/2*Sin(iAngle),iCoord1y+GroutWidth/2*Cos(iAngle),iCoord1x+GroutWidth/2*Sin(iAngle)+GroutHeight*Cos(iAngle),iCoord1y-GroutHeight*Sin(iAngle)+GroutWidth/2*Cos(iAngle),iCoord1x-GroutWidth/2*Sin(iAngle)+GroutHeight*Cos(iAngle),iCoord1y-GroutHeight*Sin(iAngle)-GroutWidth/2*Cos(iAngle);

                CASE 3:

                    IF iCoord1x-GroutWidth/2*Cos(iAngle)-GroutHeight*Sin(iAngle)<BedXmin OR iCoord1y-GroutHeight*Cos(iAngle)+GroutWidth/2*Sin(iAngle)<BedYmin OR iCoord1x-GroutWidth/2*Cos(iAngle)<BedXmin OR iCoord1y+GroutWidth/2*Sin(iAngle)<BedYmin OR iCoord1x+GroutWidth/2*Cos(iAngle)<BedXmin OR iCoord1y-GroutWidth/2*Sin(iAngle)<BedYmin OR iCoord1x+GroutWidth/2*Cos(iAngle)-GroutHeight*Sin(iAngle)<BedXmin OR iCoord1y-GroutHeight*Cos(iAngle)-GroutWidth/2*Sin(iAngle)<BedYmin OR ((iCoord1x-GroutHeight)*(iCoord1x-GroutWidth)+(iCoord1y-GroutHeight)*(iCoord1y-GroutWidth)<2560000) THEN
                        RAISE ERR_INVALID_INPUT;
                    ENDIF

                    IF iCoord1x-GroutWidth/2*Cos(iAngle)-GroutHeight*Sin(iAngle)>BedXmax OR iCoord1y-GroutHeight*Cos(iAngle)+GroutWidth/2*Sin(iAngle)>BedYmax OR iCoord1x-GroutWidth/2*Cos(iAngle)>BedXmax OR iCoord1y+GroutWidth/2*Sin(iAngle)>BedYmax OR iCoord1x+GroutWidth/2*Cos(iAngle)>BedXmax OR iCoord1y-GroutWidth/2*Sin(iAngle)>BedYmax OR iCoord1x+GroutWidth/2*Cos(iAngle)-GroutHeight*Sin(iAngle)>BedXmax OR iCoord1y-GroutHeight*Cos(iAngle)-GroutWidth/2*Sin(iAngle)>BedYmax THEN
                        RAISE ERR_INVALID_INPUT;
                    ENDIF

                    PlotRect iCoord1x-GroutWidth/2*Cos(iAngle)-GroutHeight*Sin(iAngle),iCoord1y-GroutHeight*Cos(iAngle)+GroutWidth/2*Sin(iAngle),iCoord1x-GroutWidth/2*Cos(iAngle),iCoord1y+GroutWidth/2*Sin(iAngle),iCoord1x+GroutWidth*Cos(iAngle),iCoord1y-GroutWidth/2*Sin(iAngle),iCoord1x+GroutWidth/2*Cos(iAngle)-GroutHeight*Sin(iAngle),iCoord1y-GroutHeight*Cos(iAngle)-GroutWidth/2*Sin(iAngle);


                CASE 4:

                    IF iCoord1x-GroutWidth/2*Sin(iAngle)-GroutHeight*Cos(iAngle)<BedXmin OR iCoord1y+GroutHeight*Sin(iAngle)-GroutWidth/2*Cos(iAngle)<BedYmin OR iCoord1x+GroutWidth/2*Sin(iAngle)-GroutHeight*Cos(iAngle)<BedXmin OR iCoord1y+GroutHeight*Sin(iAngle)+GroutWidth/2*Cos(iAngle)<BedYmin OR iCoord1x+GroutWidth/2*Sin(iAngle)<BedXmin OR iCoord1y+GroutWidth/2*Cos(iAngle)<BedYmin OR iCoord1x-GroutWidth/2*Sin(iAngle)<BedXmin OR iCoord1y-GroutWidth/2*Cos(iAngle)<BedYmin OR ((iCoord1x-GroutHeight)*(iCoord1x-GroutWidth)+(iCoord1y-GroutHeight)*(iCoord1y-GroutWidth)<2560000) THEN
                        RAISE ERR_INVALID_INPUT;
                    ENDIF

                    IF iCoord1x-GroutWidth/2*Sin(iAngle)-GroutHeight*Cos(iAngle)>BedXmax OR iCoord1y+GroutHeight*Sin(iAngle)-GroutWidth/2*Cos(iAngle)>BedYmax OR iCoord1x+GroutWidth/2*Sin(iAngle)-GroutHeight*Cos(iAngle)>BedXmax OR iCoord1y+GroutHeight*Sin(iAngle)+GroutWidth/2*Cos(iAngle)>BedYmax OR iCoord1x+GroutWidth/2*Sin(iAngle)>BedXmax OR iCoord1y+GroutWidth/2*Cos(iAngle)>BedYmax OR iCoord1x-GroutWidth/2*Sin(iAngle)>BedXmax OR iCoord1y-GroutWidth/2*Cos(iAngle)>BedYmax THEN
                        RAISE ERR_INVALID_INPUT;
                    ENDIF

                    PlotRect iCoord1x-GroutWidth/2*Sin(iAngle)-GroutHeight*Cos(iAngle),iCoord1y+GroutHeight*Sin(iAngle)-GroutWidth/2*Cos(iAngle),iCoord1x+GroutWidth/2*Sin(iAngle)-GroutHeight*Cos(iAngle),iCoord1y+GroutHeight*Sin(iAngle)+GroutWidth/2*Cos(iAngle),iCoord1x+GroutWidth/2*Sin(iAngle),iCoord1y+GroutWidth/2*Cos(iAngle),iCoord1x-GroutWidth/2*Sin(iAngle),iCoord1y-GroutWidth/2*Cos(iAngle);
                DEFAULT:
                    RAISE ERR_INVALID_INPUT;

                ENDTEST

            ELSEIF iPlotType=4 THEN
                ! Rectangle with cross
                TPWrite "Enter the centre coordinate";
                TPReadNum iCoord1x,"Enter centre coordinate X value";
                TPReadNum iCoord1y,"Enter centre coordinate y value";

                IF (iCoord1x-TieInWidth/2)<BedXmin OR (iCoord1y-TieInWidth/2)<BedYmin OR (iCoord1x+TieInWidth/2)>BedXmax OR (iCoord1y+TieInWidth/2)>BedYmax OR (iCoord1x*iCoord1x+iCoord1y*iCoord1y<2560000) THEN
                    RAISE ERR_INVALID_INPUT;
                ENDIF
                PlotRect iCoord1x-TieInWidth/2,iCoord1y-TieInWidth/2,iCoord1x-TieInWidth/2,iCoord1y+TieInWidth/2,iCoord1x+TieInWidth/2,iCoord1y+TieInWidth/2,iCoord1x+TieInWidth/2,iCoord1y-TieInWidth/2;
                PlotLine iCoord1x,iCoord1y-TieInWidth/2,iCoord1x,iCoord1y+TieInWidth/2;
                PlotLine iCoord1x-TieInWidth/2,iCoord1y,iCoord1x+TieInWidth/2,iCoord1y;


            ELSEIF iPlotType=5 THEN
                !triangle
                TPWrite "Enter the edge coordinate and angle";
                TPReadNum iCoord1x,"Enter centre coordinate X value";
                TPReadNum iCoord1y,"Enter centre coordinate y value";
                TPWrite "0 degrees is up, 90 is pointing right/CW, 180 pointing down, 270 pointing left.";
                TPReadNum iAngle,"Enter the angle";

                IF (iAngle>=0 AND iAngle<=45) OR (iAngle>315 AND iAngle<=360) THEN
                    TriangleAngle:=iAngle;
                    IF iCoord1x-TriangleBase/2*Cos(TriangleAngle)<BedXmin OR iCoord1y+TriangleBase/2*Sin(TriangleAngle)<BedYmin OR iCoord1x+TriangleHeight*Sin(TriangleAngle)<BedXmin OR iCoord1y+TriangleHeight*Cos(TriangleAngle)<BedYmin OR iCoord1x+TriangleBase/2*Cos(TriangleAngle)<BedXmin OR iCoord1y-TriangleBase/2*Sin(TriangleAngle)<BedYmin OR iCoord1x-TriangleBase/2*Cos(TriangleAngle)>BedXmax OR iCoord1y+TriangleBase/2*Sin(TriangleAngle)>BedYmax OR iCoord1x+TriangleHeight*Sin(TriangleAngle)>BedXmax OR iCoord1y+TriangleHeight*Cos(TriangleAngle)>BedYmax OR iCoord1x+TriangleBase/2*Cos(TriangleAngle)>BedXmax OR iCoord1y-TriangleBase/2*Sin(TriangleAngle)>BedYmax OR (iCoord1x*iCoord1x+iCoord1y*iCoord1y<2560000) THEN
                        RAISE ERR_INVALID_INPUT;
                    ENDIF
                    PlotLine iCoord1x-TriangleBase/2*Cos(TriangleAngle),iCoord1y+TriangleBase/2*Sin(TriangleAngle),iCoord1x+TriangleHeight*Sin(TriangleAngle),iCoord1y+TriangleHeight*Cos(TriangleAngle);
                    PlotLine iCoord1x+TriangleHeight*Sin(TriangleAngle),iCoord1y+TriangleHeight*Cos(TriangleAngle),iCoord1x+TriangleBase/2*Cos(TriangleAngle),iCoord1y-TriangleBase/2*Sin(TriangleAngle);
                    PlotLine iCoord1x+TriangleBase/2*Cos(TriangleAngle),iCoord1y-TriangleBase/2*Sin(TriangleAngle),iCoord1x-TriangleBase/2*Cos(TriangleAngle),iCoord1y+TriangleBase/2*Sin(TriangleAngle);

                ELSEIF iAngle<=135 AND iAngle>45 THEN
                    TriangleAngle:=iAngle-90;
                    IF iCoord1x-TriangleBase/2*Sin(TriangleAngle)<BedXmin OR iCoord1y-TriangleBase/2*Cos(TriangleAngle)<BedYmin OR iCoord1x+TriangleBase/2*Sin(TriangleAngle)<BedXmin OR iCoord1y-TriangleBase/2*Sin(TriangleAngle)<BedYmin OR iCoord1x+TriangleHeight*Cos(TriangleAngle)<BedXmin OR iCoord1y-TriangleHeight*Sin(TriangleAngle)<BedYmin OR iCoord1x-TriangleBase/2*Sin(TriangleAngle)>BedXmax OR iCoord1y-TriangleBase/2*Cos(TriangleAngle)>BedYmax OR iCoord1x+TriangleBase/2*Sin(TriangleAngle)>BedXmax OR iCoord1y-TriangleBase/2*Sin(TriangleAngle)>BedYmax OR iCoord1x+TriangleHeight*Cos(TriangleAngle)>BedXmax OR iCoord1y-TriangleHeight*Sin(TriangleAngle)>BedYmax OR (iCoord1x*iCoord1x+iCoord1y*iCoord1y<2560000) THEN

                        RAISE ERR_INVALID_INPUT;
                    ENDIF
                    PlotLine iCoord1x-TriangleBase/2*Sin(TriangleAngle),iCoord1y-TriangleBase/2*Cos(TriangleAngle),iCoord1x+TriangleBase/2*Sin(TriangleAngle),iCoord1y+TriangleBase/2*Cos(TriangleAngle);
                    PlotLine iCoord1x+TriangleBase/2*Sin(TriangleAngle),iCoord1y+TriangleBase/2*Cos(TriangleAngle),iCoord1x+TriangleHeight*Cos(TriangleAngle),iCoord1y-TriangleHeight*Sin(TriangleAngle);
                    PlotLine iCoord1x+TriangleHeight*Cos(TriangleAngle),iCoord1y-TriangleHeight*Sin(TriangleAngle),iCoord1x-TriangleBase/2*Sin(TriangleAngle),iCoord1y-TriangleBase/2*Cos(TriangleAngle);

                ELSEIF iAngle<=225 AND iAngle>135 THEN
                    TriangleAngle:=iAngle-180;
                    IF iCoord1x-TriangleHeight*Sin(TriangleAngle)<BedXmin OR iCoord1y-TriangleHeight*Sin(TriangleAngle)<BedYmin OR iCoord1x-TriangleBase/2*Cos(TriangleAngle)<BedXmin OR iCoord1y+TriangleBase/2*Sin(TriangleAngle)<BedYmin OR iCoord1x+TriangleBase/2*Cos(TriangleAngle)<BedXmin OR iCoord1y-TriangleBase/2*Sin(TriangleAngle)<BedYmin OR iCoord1x-TriangleHeight*Sin(TriangleAngle)>BedXmax OR iCoord1y-TriangleHeight*Sin(TriangleAngle)>BedYmax OR iCoord1x-TriangleBase/2*Cos(TriangleAngle)>BedXmax OR iCoord1y+TriangleBase/2*Sin(TriangleAngle)>BedYmax OR iCoord1x+TriangleBase/2*Cos(TriangleAngle)>BedXmax OR iCoord1y-TriangleBase/2*Sin(TriangleAngle)>BedYmax OR (iCoord1x*iCoord1x+iCoord1y*iCoord1y<2560000) THEN

                        RAISE ERR_INVALID_INPUT;
                    ENDIF
                    PlotLine iCoord1x-TriangleHeight*Sin(TriangleAngle),iCoord1y-TriangleHeight*Cos(TriangleAngle),iCoord1x-TriangleBase/2*Cos(TriangleAngle),iCoord1y+TriangleBase/2*Sin(TriangleAngle);
                    PlotLine iCoord1x-TriangleBase/2*Cos(TriangleAngle),iCoord1y+TriangleBase/2*Sin(TriangleAngle),iCoord1x+TriangleBase/2*Cos(TriangleAngle),iCoord1y-TriangleBase/2*Sin(TriangleAngle);
                    PlotLine iCoord1x+TriangleBase/2*Cos(TriangleAngle),iCoord1y-TriangleBase/2*Sin(TriangleAngle),iCoord1x-TriangleHeight*Sin(TriangleAngle),iCoord1y-TriangleHeight*Cos(TriangleAngle);

                ELSEIF iAngle<=315 AND iAngle>225 THEN
                    TriangleAngle:=iAngle-270;
                    IF iCoord1x-TriangleBase/2*Sin(TriangleAngle)<BedXmin OR iCoord1y-TriangleBase/2*Cos(TriangleAngle)<BedYmin OR iCoord1x+TriangleHeight*Cos(TriangleAngle)<BedXmin OR iCoord1y-TriangleHeight*Sin(TriangleAngle)<BedYmin OR iCoord1x+TriangleBase/2*Sin(TriangleAngle)<BedXmin OR iCoord1y+TriangleBase/2*Cos(TriangleAngle)<BedYmin OR iCoord1x-TriangleBase/2*Sin(TriangleAngle)>BedXmax OR iCoord1y-TriangleBase/2*Cos(TriangleAngle)>BedYmax OR iCoord1x+TriangleHeight*Cos(TriangleAngle)>BedXmax OR iCoord1y-TriangleHeight*Sin(TriangleAngle)>BedYmax OR iCoord1x+TriangleBase/2*Sin(TriangleAngle)>BedXmax OR iCoord1y+TriangleBase/2*Cos(TriangleAngle)>BedYmax OR (iCoord1x*iCoord1x+iCoord1y*iCoord1y<2560000) THEN
                        RAISE ERR_INVALID_INPUT;
                    ENDIF

                    PlotLine iCoord1x-TriangleBase/2*Sin(TriangleAngle),iCoord1y-TriangleBase/2*Cos(TriangleAngle),iCoord1x-TriangleHeight*Cos(TriangleAngle),iCoord1y+TriangleHeight*Sin(TriangleAngle);
                    PlotLine iCoord1x-TriangleHeight*Cos(TriangleAngle),iCoord1y+TriangleHeight*Sin(TriangleAngle),iCoord1x+TriangleBase/2*Sin(TriangleAngle),iCoord1y+TriangleBase/2*Cos(TriangleAngle);
                    PlotLine iCoord1x+TriangleBase/2*Sin(TriangleAngle),iCoord1y+TriangleBase/2*Cos(TriangleAngle),iCoord1x-TriangleBase/2*Sin(TriangleAngle),iCoord1y-TriangleBase/2*Cos(TriangleAngle);



                ELSE
                    RAISE ERR_INVALID_INPUT;
                ENDIF

            ELSE
                RAISE ERR_INVALID_INPUT;
            ENDIF

        CASE 4:
            TPWrite "Enter the x coordinates for the start and end positions of the formwork.";
            TPReadNum iCoord1x,"Enter first coordinate X value";
            TPReadNum iCoord2x,"Enter second coordinate x value";
            TPReadNum iZoffset,"Enter Z offset (-ve for lower, +ve for higher, 0 for no change:";
            IF iCoord1x<0 OR iCoord2x<0 OR iCoord1x>7900 OR iCoord2x>7900 THEN
                RAISE ERR_INVALID_INPUT;
            ENDIF

            IF iCoord1x>iCoord2x THEN
                iCoordTemp:=iCoord1x;
                iCoord1x:=iCoord2x;
                iCoord2x:=iCoordTemp;
            ENDIF

            Screed iCoord1x,iCoord2x,iZoffset,11;

        CASE 5:
            TPWrite "Enter the coordinates for the corner closest to the robot home position.";
            TPReadNum iCoord1x,"Enter first coordinate X value";
            TPReadNum iCoord1y,"Enter first coordinate y value";
            TPWrite "Enter the coordinates for the corner furthest from the robot home position.";
            TPReadNum iCoord2x,"Enter second coordinate X value";
            TPReadNum iCoord2y,"Enter second coordinate y value";
            TPReadNum iHeliBladeSpeed,"Enter speed of heli blades (rpm from 0 - 140).";
            TPReadNum iHeliBladeAngle,"Enter heli blade angle (degrees from 0 - 12).";
            TPReadNum iZoffset,"Enter Z offset (-ve for lower, +ve for higher, 0 for no change:";
            TPReadNum iHeliPan,"Enter 1 for pan attachment or 2 for just blades:";
            !TPReadNum iLRUD,"Enter 1 for left/right movement or 2 for up/down movement:";

            IF iCoord1x<0 OR iCoord1y<0 OR iCoord2x<0 OR iCoord2y<0 OR iCoord1x>8800 OR iCoord1y>2400 OR iCoord2x>8800 OR iCoord2y>2400 OR iHeliBladeSpeed<0 OR iHeliBladeSpeed>140 OR iHeliBladeAngle<0 OR iHeliBladeAngle>12 OR iCoord2y<iCoord1y OR iCoord2x<iCoord1x OR iHeliPan<1 OR iHeliPan>2 THEN
                RAISE ERR_INVALID_INPUT;
            ENDIF
            !IF iLRUD=1 THEN
            HeliTrowelLR iCoord1x,iCoord1y,iCoord2x,iCoord2y,iHeliBladeSpeed,iHeliBladeAngle,iZoffset,iHeliPan;
            !ELSEIF iLRUD=2 THEN
            !    HeliTrowelUD iCoord1x,iCoord1y,iCoord2x,iCoord2y,iHeliBladeSpeed,iHeliBladeAngle,iZoffset,iHeliPan;
            !ELSE
            !    RAISE ERR_INVALID_INPUT;
            !ENDIF

        CASE 6:
            VacuumBed;

        CASE 7:
            Polish;
        DEFAULT:
            RAISE ERR_INVALID_INPUT;
        ENDTEST
    ERROR
        RAISE ;
    ENDPROC

    PROC HeliTrowelLR(num HeliStartX,num HeliStartY,num HeliEndX,num HeliEndY,num HeliSpeed,num HeliAngle,num HeliZoffset,num IsPan)

        pHeliStart.trans:=[HeliStartX,HeliStartY,(FormHeight+HeliZoffset)];
        pHeliEnd.trans:=[HeliEndX,HeliEndY,(FormHeight+HeliZoffset)];

        IF ToolNum<>2 THEN
            Home;
            Heli_Pickup;
        ENDIF

        IF pHeliStart.trans.y<1800 THEN
            pHeliStart.extax.eax_a:=Bed1Wyong.uframe.trans.x-pHeliStart.trans.x+1000+HeliBladeWidth/2;
            pHeliEnd.extax.eax_a:=Bed1Wyong.uframe.trans.x-pHeliEnd.trans.x+1000-HeliBladeWidth/2;
        ELSE
            pHeliStart.extax.eax_a:=Bed1Wyong.uframe.trans.x-pHeliStart.trans.x+HeliBladeWidth/2;
            pHeliEnd.extax.eax_a:=Bed1Wyong.uframe.trans.x-pHeliEnd.trans.x-HeliBladeWidth/2;
        ENDIF

        IF (pHeliEnd.trans.y-pHeliStart.trans.y)<HeliBladeWidth THEN
            HeliPasses:=1;
            HeliPassWidth:=0;
        ELSE
            HeliPasses:=((pHeliEnd.trans.y-pHeliStart.trans.y-HeliBladeWidth) DIV HeliOverlapMin);
            IF HeliPasses MOD 2<>0 THEN
                Incr HeliPasses;
            ENDIF
            IF HeliPasses<1 THEN
                HeliPasses:=1;
            ENDIF
            HeliPassWidth:=(pHeliEnd.trans.y-(HeliBladeWidth/2)-(pHeliStart.trans.y+(HeliBladeWidth/2)))/HeliPasses;
        ENDIF

        pHeliTempS:=pHeliStart;
        pHeliTempE:=pHeliEnd;
        pHeliTempS.trans.x:=pHeliStart.trans.x-(HeliBladeWidth/2)+300;
        pHeliTempS.trans.y:=pHeliStart.trans.y+(HeliBladeWidth/2);
        pHeliTempE.trans.x:=pHeliEnd.trans.x-(HeliBladeWidth/2)-300;
        pHeliTempE.trans.y:=pHeliEnd.trans.y-(HeliBladeWidth/2);
        pHeliTempS.trans.z:=FormHeight+HeliZoffset;
        pHeliTempE.trans.z:=FormHeight+HeliZoffset;

        MoveJ Offs(pHeliTempS,0,0,300),v500,z5,tHeli\WObj:=Bed1Wyong;

        IF IsPan=2 THEN
            HeliBlade_Angle HeliAngle;
            HeliBladeSpeed HeliSpeed,"FWD";
            WaitTime\inpos,4;
        ENDIF

        IF IsPan=1 THEN
            MoveJ Offs(pHeliTempS,0,0,75),v500,z5,tHeli\WObj:=Bed1Wyong;
            Stop;
        ENDIF
        HeliZ pHeliTempS.trans.x,pHeliTempS.trans.y,TRUE;
        HeliZOffs:=HighestArray(HeliZArrayCounter);

        MoveL Offs(pHeliTempS,0,0,PitchZOffset+HeliZOffs),v50,z5,tHeli\WObj:=Bed1Wyong;
        pHeliTemp1:=pHeliTempS;
        pHeliTemp2:=pHeliTempS;
        pHeliTemp2.trans.x:=pHeliTempE.trans.x;
        pHeliTemp2.extax.eax_a:=pHeliTempE.extax.eax_a;

        IF IsPan=1 THEN
            Stop;
            HeliBlade_Angle HeliAngle;
            HeliBladeSpeed HeliSpeed,"FWD";
            WaitTime\inpos,5;
        ENDIF

        HeliDiv:=(pHeliTempE.trans.x-pHeliTempS.trans.x) DIV XGridSpacing;

        FOR i FROM 0 to (2*HeliPasses) DO
            IF (i MOD 2)=0 THEN

                !Needs fixing of -1*x
                FOR M FROM 0 TO (HeliDiv-1) DO
                    HeliZ(pHeliTemp1.trans.x-M*XGridSpacing+XGridSpacing),(pHeliTemp1.trans.y+HeliPassWidth*i/2),TRUE;
                    HeliZOffs:=HighestArray(HeliZArrayCounter);
                    IF (HeliPassWidth*i/2+pHeliTemp1.trans.y)>1600 THEN
                        pHeliTemp1.extax.eax_a:=pHeliTemp1.trans.x+Bed1Wyong.uframe.trans.x-M*XGridSpacing;
                    ELSE
                        pHeliTemp1.extax.eax_a:=pHeliTemp1.trans.x+Bed1Wyong.uframe.trans.x+1000-M*XGridSpacing;
                    ENDIF
                    MoveL Offs(pHeliTemp1,-1*M*XGridSpacing,HeliPassWidth*i/2,PitchZOffset+HeliZOffs),vHeli,z5,tHeli\WObj:=Bed1Wyong;
                    !Across Right
                ENDFOR

                IF (HeliPassWidth*i/2+pHeliTemp2.trans.y)>1600 THEN
                    pHeliTemp2.extax.eax_a:=pHeliTemp2.trans.x+Bed1Wyong.uframe.trans.x;
                ELSE
                    pHeliTemp2.extax.eax_a:=pHeliTemp2.trans.x+Bed1Wyong.uframe.trans.x+1000;
                ENDIF
                HeliZ(pHeliTemp2.trans.x),(pHeliTemp1.trans.y+HeliPassWidth*i/2),TRUE;
                HeliZOffs:=HighestArray(HeliZArrayCounter);
                MoveL Offs(pHeliTemp2,0,HeliPassWidth*i/2,PitchZOffset+HeliZOffs),vHeli,z5,tHeli\WObj:=Bed1Wyong;
                !Across Right

                IF i=(2*HeliPasses) THEN
                ELSE
                    HeliZ(pHeliTemp2.trans.x),(pHeliTemp1.trans.y+HeliPassWidth*(i+1)/2),TRUE;
                    HeliZOffs:=HighestArray(HeliZArrayCounter);
                    IF (HeliPassWidth*(i+1)/2+pHeliTemp2.trans.y)>1600 THEN
                        pHeliTemp2.extax.eax_a:=pHeliTemp2.trans.x+Bed1Wyong.uframe.trans.x;
                    ELSE
                        pHeliTemp2.extax.eax_a:=pHeliTemp2.trans.x+Bed1Wyong.uframe.trans.x+1000;
                    ENDIF
                    MoveL Offs(pHeliTemp2,0,HeliPassWidth*(i+1)/2,PitchZOffset+HeliZOffs),vHeli,z5,tHeli\WObj:=Bed1Wyong;
                    !Up

                    FOR M FROM (HeliDiv-1) TO 0 DO
                        HeliZ(pHeliTemp1.trans.x-M*XGridSpacing),(pHeliTemp1.trans.y+HeliPassWidth*(i+1)/2),TRUE;
                        HeliZOffs:=HighestArray(HeliZArrayCounter);
                        IF (HeliPassWidth*(i+1)/2+pHeliTemp1.trans.y)>1600 THEN
                            pHeliTemp1.extax.eax_a:=pHeliTemp1.trans.x+Bed1Wyong.uframe.trans.x-M*XGridSpacing;
                        ELSE
                            pHeliTemp1.extax.eax_a:=pHeliTemp1.trans.x+Bed1Wyong.uframe.trans.x+1000-M*XGridSpacing;
                        ENDIF
                        MoveL Offs(pHeliTemp1,-1*M*XGridSpacing,HeliPassWidth*(i+1)/2,PitchZOffset+HeliZOffs),vHeli,z5,tHeli\WObj:=Bed1Wyong;
                        !Across Left
                    ENDFOR

                ENDIF

            ENDIF
        ENDFOR

        IF IsPan=1 THEN
            WaitTime\InPos,0.1;
            HeliBladeSpeed 0,"FWD";
            WaitTime\inpos,8;
            MoveL Offs(pHeliTemp2,0,HeliPassWidth*2*HeliPasses/2,18+PitchZOffset+HeliZOffs),v50,fine,tHeli\WObj:=Bed1Wyong;
            HeliBladeSpeed 20,"REV";
            WaitTime\inpos,0.6;
            HeliBladeSpeed 0,"FWD";
            Stop;
        ENDIF
        MoveL Offs(pHeliTemp2,0,HeliPassWidth*2*HeliPasses/2,50+PitchZOffset+HeliZOffs),v50,z5,tHeli\WObj:=Bed1Wyong;

        HeliBladeSpeed 0,"FWD";
        CurrentJoints:=CJointT();
        CurrentPos:=CalcRobT(CurrentJoints,tHeli\WObj:=wobj0);
        MoveJ Offs(pHeliTemp2,0,2500-CurrentPos.trans.y,300),v500,z5,tHeli\WObj:=Bed1Wyong;
        MoveJ Offs(ptHeli,0,0,500),v500,fine,tHeli;

    ENDPROC

    PROC HeliPanLR(num HeliStartX,num HeliStartY,num HeliEndX,num HeliEndY,speeddata HeliVTCP,num HeliSpeed,num HeliZoffset)

        pHeliStart.trans:=[-1*HeliStartX,HeliStartY,(FormHeight+14+HeliZoffset)];
        pHeliEnd.trans:=[-1*HeliEndX,HeliEndY,(FormHeight+14+HeliZoffset)];

        IF ToolNum<>2 THEN
            Home;
            Heli_Pickup;
        ELSE
            pTemp:=ptHeli;
            pTemp.extax.eax_a:=ptHeli.extax.eax_a-2000;
            pTemp.trans.z:=ptHeli.trans.z+800;
            MoveJ Offs(pTemp,-2000,0,0),v500,fine,tHeli;
        ENDIF

        IF pHeliStart.trans.y<1800 THEN
            pHeliStart.extax.eax_a:=Bed1Wyong.uframe.trans.x+pHeliStart.trans.x+1000+HeliBladeWidth/2;
            pHeliEnd.extax.eax_a:=Bed1Wyong.uframe.trans.x+pHeliEnd.trans.x+1000-HeliBladeWidth/2;
        ELSE
            pHeliStart.extax.eax_a:=Bed1Wyong.uframe.trans.x+pHeliStart.trans.x+HeliBladeWidth/2;
            pHeliEnd.extax.eax_a:=Bed1Wyong.uframe.trans.x+pHeliEnd.trans.x-HeliBladeWidth/2;
        ENDIF

        IF (pHeliEnd.trans.y-pHeliStart.trans.y)<HeliBladeWidth THEN
            HeliPasses:=1;
            HeliPassWidth:=0;
        ELSE
            HeliPasses:=((pHeliEnd.trans.y-pHeliStart.trans.y-HeliBladeWidth) DIV PanOverlapMin);
            IF HeliPasses MOD 2<>0 THEN
                Incr HeliPasses;
            ENDIF
            IF HeliPasses<1 THEN
                HeliPasses:=1;
            ENDIF
            HeliPassWidth:=(pHeliEnd.trans.y-(HeliBladeWidth/2)-(pHeliStart.trans.y+(HeliBladeWidth/2)))/HeliPasses;
        ENDIF

        pHeliTempS:=pHeliStart;
        pHeliTempE:=pHeliEnd;
        pHeliTempS.trans.x:=pHeliStart.trans.x+(HeliBladeWidth/2)-300;
        pHeliTempS.trans.y:=pHeliStart.trans.y+(HeliBladeWidth/2);
        pHeliTempE.trans.x:=pHeliEnd.trans.x-(HeliBladeWidth/2)+300;
        pHeliTempE.trans.y:=pHeliEnd.trans.y-(HeliBladeWidth/2);
        pHeliTempS.trans.z:=FormHeight+HeliZoffset;
        pHeliTempE.trans.z:=FormHeight+HeliZoffset;

        MoveJ Offs(pHeliTempS,0,0,300),v500,z5,tHeli\WObj:=Bed1Wyong;

        MoveJ Offs(pHeliTempS,0,0,75),v500,z5,tHeli\WObj:=Bed1Wyong;
        TPWrite "Place pan under blades.";
        Stop;

        HeliZ pHeliTempS.trans.x,pHeliTempS.trans.y,TRUE;
        HeliZOffs:=HighestArray(HeliZArrayCounter);

        MoveL Offs(pHeliTempS,0,0,PitchZOffset+HeliZOffs),v50,z5,tHeli\WObj:=Bed1Wyong;
        pHeliTemp1:=pHeliTempS;
        pHeliTemp2:=pHeliTempS;
        pHeliTemp2.trans.x:=pHeliTempE.trans.x;
        pHeliTemp2.extax.eax_a:=pHeliTempE.extax.eax_a;

        TPWrite "Check blades are under tabs plane";
        Stop;
        HeliBlade_Angle 0;
        HeliBladeSpeed HeliSpeed,"FWD";
        WaitTime\inpos,5;

        HeliDiv:=(abs(pHeliTempE.trans.x)-abs(pHeliTempS.trans.x)) DIV XGridSpacing;

        FOR i FROM 0 to (2*HeliPasses) DO
            IF (i MOD 2)=0 THEN


                FOR M FROM 0 TO (HeliDiv-1) DO
                    HeliZ(pHeliTemp1.trans.x-M*XGridSpacing-XGridSpacing),(pHeliTemp1.trans.y+HeliPassWidth*i/2),TRUE;
                    HeliZOffs:=HighestArray(HeliZArrayCounter);
                    IF (HeliPassWidth*i/2+pHeliTemp1.trans.y)>1600 THEN
                        pHeliTemp1.extax.eax_a:=Bed1Wyong.uframe.trans.x+pHeliTemp1.trans.x-M*XGridSpacing;
                    ELSE
                        pHeliTemp1.extax.eax_a:=Bed1Wyong.uframe.trans.x+pHeliTemp1.trans.x+1000-M*XGridSpacing;
                    ENDIF
                    MoveL Offs(pHeliTemp1,-1*M*XGridSpacing,HeliPassWidth*i/2,PitchZOffset+HeliZOffs),HeliVTCP,z5,tHeli\WObj:=Bed1Wyong;
                    !Across Left
                ENDFOR

                IF (HeliPassWidth*i/2+pHeliTemp2.trans.y)>1600 THEN
                    pHeliTemp2.extax.eax_a:=Bed1Wyong.uframe.trans.x+pHeliTemp2.trans.x;
                ELSE
                    pHeliTemp2.extax.eax_a:=Bed1Wyong.uframe.trans.x+pHeliTemp2.trans.x+1000;
                ENDIF
                HeliZ(pHeliTemp2.trans.x),(pHeliTemp1.trans.y+HeliPassWidth*i/2),TRUE;
                HeliZOffs:=HighestArray(HeliZArrayCounter);
                MoveL Offs(pHeliTemp2,0,HeliPassWidth*i/2,PitchZOffset+HeliZOffs),HeliVTCP,z5,tHeli\WObj:=Bed1Wyong;
                !Across Left final position

                IF i=(2*HeliPasses) THEN
                ELSE
                    HeliZ(pHeliTemp2.trans.x),(pHeliTemp1.trans.y+HeliPassWidth*(i+1)/2),TRUE;
                    HeliZOffs:=HighestArray(HeliZArrayCounter);
                    IF (HeliPassWidth*(i+1)/2+pHeliTemp2.trans.y)>1600 THEN
                        pHeliTemp2.extax.eax_a:=Bed1Wyong.uframe.trans.x+pHeliTemp2.trans.x;
                    ELSE
                        pHeliTemp2.extax.eax_a:=Bed1Wyong.uframe.trans.x+pHeliTemp2.trans.x+1000;
                    ENDIF
                    MoveL Offs(pHeliTemp2,0,HeliPassWidth*(i+1)/2,PitchZOffset+HeliZOffs),HeliVTCP,z5,tHeli\WObj:=Bed1Wyong;
                    !Up

                    FOR M FROM (HeliDiv-1) TO 0 DO
                        HeliZ(pHeliTemp1.trans.x-M*XGridSpacing),(pHeliTemp1.trans.y+HeliPassWidth*(i+1)/2),TRUE;
                        HeliZOffs:=HighestArray(HeliZArrayCounter);
                        IF (HeliPassWidth*(i+1)/2+pHeliTemp1.trans.y)>1600 THEN
                            pHeliTemp1.extax.eax_a:=Bed1Wyong.uframe.trans.x+pHeliTemp1.trans.x-M*XGridSpacing;
                        ELSE
                            pHeliTemp1.extax.eax_a:=Bed1Wyong.uframe.trans.x+pHeliTemp1.trans.x+1000-M*XGridSpacing;
                        ENDIF
                        MoveL Offs(pHeliTemp1,-1*M*XGridSpacing,HeliPassWidth*(i+1)/2,PitchZOffset+HeliZOffs),HeliVTCP,z5,tHeli\WObj:=Bed1Wyong;
                        !Across Right
                    ENDFOR

                ENDIF

            ENDIF
        ENDFOR


        WaitTime\InPos,0.1;
        HeliBladeSpeed 0,"FWD";
        WaitTime\inpos,8;
        MoveL Offs(pHeliTemp2,0,HeliPassWidth*2*HeliPasses/2,18+PitchZOffset+HeliZOffs),v50,fine,tHeli\WObj:=Bed1Wyong;
        HeliBladeSpeed 20,"REV";
        WaitTime\inpos,0.6;
        HeliBladeSpeed 0,"FWD";
        TPWrite "Check pan is dettached.";
        Stop;


        MoveL Offs(pHeliTemp2,0,HeliPassWidth*2*HeliPasses/2,50+PitchZOffset+HeliZOffs),v50,z5,tHeli\WObj:=Bed1Wyong;

        HeliBladeSpeed 0,"FWD";
        pTemp:=ptHeli;
        pTemp.extax.eax_a:=ptHeli.extax.eax_a-2000;
        pTemp.trans.z:=ptHeli.trans.z+500;
        MoveJ Offs(pTemp,-2000,0,0),v500,fine,tHeli;
        CurrentJoints:=CJointT();
        CurrentJoints:=CJointT();
        CurrentPos:=CalcRobT(CurrentJoints,tHeli\WObj:=wobj0);
        MoveJ Offs(pHeliTemp2,0,2500-CurrentPos.trans.y,300),v500,z5,tHeli\WObj:=Bed1Wyong;
        TPWrite "Clean off pan.";
        Stop;

    ENDPROC

    PROC HeliTrowelUD(num HeliStartX,num HeliStartY,num HeliEndX,num HeliEndY,num HeliSpeed,num HeliAngle,num HeliZoffset,num IsPan)

        pHeliStart.trans:=[-1*HeliStartX,HeliStartY,(FormHeight+30+HeliZoffset)];
        pHeliEnd.trans:=[-1*HeliEndX,HeliEndY,(FormHeight+30+HeliZoffset)];

        IF ToolNum<>2 THEN
            Home;
            Heli_Pickup;
        ENDIF

        IF pHeliStart.trans.y<1600 THEN
            pHeliStart.extax.eax_a:=pHeliStart.trans.x+Bed1Wyong.uframe.trans.x+1000+HeliBladeWidth/2;
            pHeliEnd.extax.eax_a:=pHeliEnd.trans.x+Bed1Wyong.uframe.trans.x+1000+HeliBladeWidth/2;
        ELSE
            pHeliStart.extax.eax_a:=pHeliStart.trans.x+Bed1Wyong.uframe.trans.x+HeliBladeWidth/2;
            pHeliEnd.extax.eax_a:=pHeliEnd.trans.x+Bed1Wyong.uframe.trans.x+HeliBladeWidth/2;
        ENDIF


        IF (abs(pHeliEnd.trans.x)-abs(pHeliStart.trans.x))<HeliBladeWidth THEN
            HeliPasses:=1;
            HeliPassWidth:=0;
        ELSE
            HeliPasses:=((abs(pHeliEnd.trans.x)-abs(pHeliStart.trans.x)-HeliBladeWidth) DIV HeliOverlapMin);
            IF HeliPasses MOD 2<>0 THEN
                Incr HeliPasses;
            ENDIF
            IF HeliPasses<1 THEN
                HeliPasses:=1;
            ENDIF
            HeliPassWidth:=(abs(pHeliEnd.trans.x)-(abs(pHeliStart.trans.x))-HeliBladeWidth)/HeliPasses;
        ENDIF

        pHeliTempS:=pHeliStart;
        pHeliTempE:=pHeliEnd;
        pHeliTempS.trans.x:=pHeliStart.trans.x-(HeliBladeWidth/2)+300;
        pHeliTempS.trans.y:=pHeliStart.trans.y+(HeliBladeWidth/2);
        pHeliTempE.trans.x:=pHeliEnd.trans.x+(HeliBladeWidth/2)-300;
        pHeliTempE.trans.y:=pHeliEnd.trans.y-(HeliBladeWidth/2);
        pHeliTempS.trans.z:=FormHeight+30+HeliZoffset;
        pHeliTempE.trans.z:=FormHeight+30+HeliZoffset;

        MoveJ Offs(pHeliTempS,0,0,300),v500,z5,tHeli\WObj:=Bed1Wyong;

        IF IsPan=2 THEN
            HeliBlade_Angle HeliAngle;
            HeliBladeSpeed HeliSpeed,"FWD";
            WaitTime\inpos,4;
        ENDIF

        IF IsPan=1 THEN
            MoveJ Offs(pHeliTempS,0,0,75),v500,z5,tHeli\WObj:=Bed1Wyong;
            Stop;
        ENDIF
        HeliZ pHeliTempS.trans.x,pHeliTempS.trans.y,TRUE;
        HeliZOffs:=HighestArray(HeliZArrayCounter);

        MoveL Offs(pHeliTempS,0,0,PitchZOffset+HeliZOffs),v50,z5,tHeli\WObj:=Bed1Wyong;
        pHeliTemp1:=pHeliTempS;
        pHeliTemp2:=pHeliTempS;
        pHeliTemp2.trans.y:=pHeliTempE.trans.y;
        pHeliTemp2.extax.eax_a:=pHeliTempE.extax.eax_a;

        IF IsPan=1 THEN
            HeliBlade_Angle HeliAngle;
            HeliBladeSpeed HeliSpeed,"FWD";
            WaitTime\inpos,5;
        ENDIF


        HeliDiv:=(pHeliTempE.trans.y-pHeliTempS.trans.y) DIV YGridSpacing;


        FOR i FROM 0 to (HeliPasses) DO

            FOR M FROM 0 TO (HeliDiv-1) DO
                HeliZ(pHeliTemp1.trans.x-HeliPassWidth*i),(pHeliTemp1.trans.y+M*YGridSpacing+YGridSpacing),TRUE;
                HeliZOffs:=HighestArray(HeliZArrayCounter);
                IF (pHeliTemp1.trans.y+M*YGridSpacing+YGridSpacing)>1600 THEN
                    pHeliTemp1.extax.eax_a:=pHeliTemp1.trans.x-1*HeliPassWidth*i+Bed1Wyong.uframe.trans.x;
                ELSE
                    pHeliTemp1.extax.eax_a:=pHeliTemp1.trans.x-1*HeliPassWidth*i+Bed1Wyong.uframe.trans.x+1000;
                ENDIF
                MoveL Offs(pHeliTemp1,-1*HeliPassWidth*i,M*YGridSpacing,PitchZOffset+HeliZOffs),vHeli,z5,tHeli\WObj:=Bed1Wyong;
                !Up
            ENDFOR

            IF (pHeliTemp2.trans.y)>1600 THEN
                pHeliTemp2.extax.eax_a:=pHeliTemp2.trans.x-1*HeliPassWidth*i+Bed1Wyong.uframe.trans.x;
            ELSE
                pHeliTemp2.extax.eax_a:=pHeliTemp2.trans.x-1*HeliPassWidth*i+Bed1Wyong.uframe.trans.x+1000;
            ENDIF
            HeliZ(pHeliTemp2.trans.x),(pHeliTemp1.trans.y+HeliPassWidth*i/2),TRUE;
            HeliZOffs:=HighestArray(HeliZArrayCounter);
            MoveL Offs(pHeliTemp2,-1*HeliPassWidth*i,0,PitchZOffset+HeliZOffs),vHeli,z5,tHeli\WObj:=Bed1Wyong;
            !Up

            IF i=HeliPasses THEN
            ELSE
                HeliZ(pHeliTemp2.trans.x-HeliPassWidth*(i+1)),(pHeliTemp1.trans.y),TRUE;
                HeliZOffs:=HighestArray(HeliZArrayCounter);
                IF (pHeliTemp2.trans.y)>1600 THEN
                    pHeliTemp2.extax.eax_a:=pHeliTemp2.trans.x-1*HeliPassWidth*(i+1)+Bed1Wyong.uframe.trans.x;
                ELSE
                    pHeliTemp2.extax.eax_a:=pHeliTemp2.trans.x-1*HeliPassWidth*(i+1)+Bed1Wyong.uframe.trans.x+1000;
                ENDIF
                MoveL Offs(pHeliTemp2,-1*HeliPassWidth*(i+1),0,PitchZOffset+HeliZOffs),vHeli,z5,tHeli\WObj:=Bed1Wyong;
                !Right

                FOR M FROM (HeliDiv-1) TO 0 DO
                    HeliZ(pHeliTemp1.trans.x-HeliPassWidth*(i+1)),(pHeliTemp1.trans.y+M*YGridSpacing),TRUE;
                    HeliZOffs:=HighestArray(HeliZArrayCounter);
                    IF (pHeliTemp1.trans.y+M*YGridSpacing)>1600 THEN
                        pHeliTemp1.extax.eax_a:=pHeliTemp1.trans.x-1*HeliPassWidth*(i+1)+Bed1Wyong.uframe.trans.x;
                    ELSE
                        pHeliTemp1.extax.eax_a:=pHeliTemp1.trans.x-1*HeliPassWidth*(i+1)+Bed1Wyong.uframe.trans.x+1000;
                    ENDIF
                    MoveL Offs(pHeliTemp1,-1*HeliPassWidth*(i+1),M*YGridSpacing,PitchZOffset+HeliZOffs),vHeli,z5,tHeli\WObj:=Bed1Wyong;
                    !Down
                ENDFOR

            ENDIF

        ENDFOR

        IF IsPan=1 THEN
            WaitTime\InPos,0.1;
            HeliBladeSpeed 0,"FWD";
            WaitTime\inpos,8;
            MoveL Offs(pHeliTemp2,HeliPassWidth*(2*HeliPasses)/2,0,18+PitchZOffset+HeliZOffs),v50,fine,tHeli\WObj:=Bed1Wyong;
            HeliBladeSpeed 20,"REV";
            WaitTime\inpos,0.6;
            HeliBladeSpeed 0,"FWD";
            Stop;
        ENDIF
        MoveL Offs(pHeliTemp2,HeliPassWidth*2*HeliPasses/2,0,50+PitchZOffset+HeliZOffs),v50,z5,tHeli\WObj:=Bed1Wyong;

        HeliBladeSpeed 0,"FWD";
        CurrentJoints:=CJointT();
        CurrentPos:=CalcRobT(CurrentJoints,tHeli\WObj:=wobj0);
        MoveL Offs(pHeliTemp2,HeliPassWidth*(2*HeliPasses)/2,2000-CurrentPos.trans.y,300),v500,z5,tHeli\WObj:=Bed1Wyong;
        MoveJ Offs(ptHeli,0,0,500),v500,z5,tHeli;

    ENDPROC

    PROC Screed(num ScrStart,num ScrEnd,num ScrZoffset,num ScrAoffset)
        VAR num StartOffset;
        VAR num EndOffset;
        CurrentJoints:=CJointT();
        CurrentPos:=CalcRobT(CurrentJoints,tVS\WObj:=Bed1Wyong);
        IF ToolNum<>3 THEN
            Home;
            VS_Pickup;
        ELSEIF (CurrentPos.trans.z<800) THEN
            MoveL Offs(CurrentPos,0,0,(800-CurrentPos.trans.z)),v200,z5,tVS\WObj:=Bed1Wyong;
        ENDIF

        StartOffset:=((pVSend.trans.z-pVSstart.trans.z)/(pVSend.trans.x-pVSstart.trans.x))*((-1*ScrStart-pVSstart.trans.x));
        EndOffset:=((pVSend.trans.z-pVSstart.trans.z)/(pVSend.trans.x-pVSstart.trans.x))*((-1*ScrEnd-pVSstart.trans.x));


        pScreedStart.trans:=[(-1*ScrStart),1910,pVSstart.trans.z+ScrZoffset+StartOffset];
        pScreedEnd.trans:=[(-1*ScrEnd),1910,pVSstart.trans.z+ScrZoffset+EndOffset];

        pScreedStart.rot:=pVSstart.rot;
        pScreedEnd.rot:=pVSend.rot;

        pScreedStart.extax.eax_a:=pScreedStart.trans.x+Bed1Wyong.uframe.trans.x+700;
        pScreedEnd.extax.eax_a:=pScreedEnd.trans.x+Bed1Wyong.uframe.trans.x+700;

        !        ScrInitialD:=(pScreedStart.trans.x) MOD 1000;
        !        IF ScrInitialD>350 AND ScrInitialD<=850 THEN
        !            ScrInitialD:=850-ScrInitialD;
        !        ELSEIF ScrInitialD>850 THEN
        !            ScrInitialD:=1000-ScrInitialD+350;
        !        ELSE
        !            ScrInitialD:=350-ScrInitialD;
        !        ENDIF

        !        IF pScreedStart.trans.x<350 THEN
        !            SStartdiv:=1;
        !            ScrBedZ:=BedZreads{1,1};
        !            pScreedStart.trans.z:=pScreedStart.trans.z+ScrBedZ;
        !        ELSEIF pScreedStart.trans.x<BedZpos{1,18,1} THEN
        !            SStartdiv:=(pScreedStart.trans.x+ScrInitialD-BedZpos{1,1,1}) DIV 500;
        !            ScrBedZ:=BedZreads{1,SStartdiv}*(1-Abs(pScreedStart.trans.x-BedZpos{1,SStartdiv,1})/500)+BedZreads{1,SStartdiv+1}*(1-Abs(pScreedStart.trans.x-BedZpos{1,SStartdiv,1+1})/500);
        !            pScreedStart.trans.z:=pScreedStart.trans.z+ScrBedZ;
        !        ELSE
        !            SStartdiv:=18;
        !            ScrBedZ:=BedZreads{1,18};
        !            pScreedStart.trans.z:=pScreedStart.trans.z+ScrBedZ;
        !        ENDIF


        !        IF pScreedEnd.trans.x<350 THEN
        !            SEnddiv:=1;
        !            ScrBedZ:=BedZreads{1,1};
        !            pScreedEnd.trans.z:=pScreedEnd.trans.z+ScrBedZ;
        !        ELSEIF pScreedEnd.trans.x<BedZpos{1,18,1} THEN
        !            SEnddiv:=(pScreedEnd.trans.x-(pScreedStart.trans.x+ScrInitialD)) DIV 500;
        !            ScrBedZ:=BedZreads{1,SEnddiv+SStartdiv}*(1-Abs(pScreedEnd.trans.x-BedZpos{1,SEnddiv+SStartdiv,1})/500)+BedZreads{1,SEnddiv+SStartdiv-1}*(1-Abs(pScreedEnd.trans.x-BedZpos{1,SEnddiv+SStartdiv-1,1})/500);
        !            pScreedEnd.trans.z:=pScreedEnd.trans.z+ScrBedZ;
        !        ELSE
        !            ScrBedZ:=BedZreads{1,18};
        !            SEnddiv:=18;
        !            pScreedEnd.trans.z:=pScreedEnd.trans.z+ScrBedZ;
        !        ENDIF

        !        MoveJ Offs(pScreedStart,-20,0,100),v1000,z5,tVS\WObj:=Bed1;
        !        VS_on;
        !        MoveL Offs(pScreedStart,-20,0,0),v100,z5,tVS\WObj:=Bed1;

        !        pScreedStart.extax.eax_a:=pScreedStart.extax.eax_a+ScrInitialD;
        !        MoveL Offs(pScreedStart,(ScrInitialD),0,BedZreads{1,(SStartdiv)}),vVS,z5,tVS\WObj:=Bed1;

        !        FOR i FROM (SStartdiv+1) TO (SEnddiv+SStartdiv) DO
        !            pScreedStart.extax.eax_a:=pScreedStart.extax.eax_a+500;
        !            MoveL Offs(pScreedStart,((i+1-(SStartdiv+1))*500+ScrInitialD),0,BedZreads{1,(i+1)}),vVS,z5,tVS\WObj:=Bed1;
        !        ENDFOR

        MoveL Offs(pScreedStart,100,0,800),v500,fine,tVS\WObj:=Bed1Wyong;
        MoveL Offs(RelTool(pScreedStart,0,0,0\Ry:=ScrAoffset),50,0,100),v500,fine,tVS\WObj:=Bed1Wyong;
        VS_on;
        MoveL Offs(RelTool(pScreedStart,0,0,0\Ry:=ScrAoffset),20,0,0),v50,z5,tVS\WObj:=Bed1Wyong;
        MoveL Offs(RelTool(pScreedEnd,0,0,0\Ry:=ScrAoffset),-140,0,0),vVS,z5,tVS\WObj:=Bed1Wyong;
        MoveL Offs(RelTool(pScreedEnd,0,0,0\Ry:=ScrAoffset),-140,0,100),v100,z5,tVS\WObj:=Bed1Wyong;
        VS_off;

        VS_Dropoff;

    ENDPROC

    PROC PlotRect(num Xcord1,num Ycord1,num Xcord2,num Ycord2,num Xcord3,num Ycord3,num Xcord4,num Ycord4)


        IF ToolNum<>4 THEN
            Home;
            Plotter_Pickup;
        ELSE
            !Check position and move to safe position if needed
            CurrentJoints:=CJointT();
            CurrentPos:=CalcRobT(CurrentJoints,tPlotter\WObj:=Bed1Wyong);

            IF (CurrentPos.trans.z<(Bed1Wyong.uframe.trans.z-30)) OR (((CurrentPos.trans.x+CurrentPos.extax.eax_a)>Bed1Wyong.uframe.trans.x) AND CurrentPos.trans.z<300) THEN
                !Robot in TS
                TPWrite("Jog robot out of tool station AND HOME");
                Stop;
            ENDIF
        ENDIF

        Plotterp1.trans:=[-1*Xcord1,Ycord1,PlotterZ];
        Plotterp2.trans:=[-1*Xcord2,Ycord2,PlotterZ];
        Plotterp3.trans:=[-1*Xcord3,Ycord3,PlotterZ];
        Plotterp4.trans:=[-1*Xcord4,Ycord4,PlotterZ];

        IF Plotterp1.trans.y>0 THEN
            IF Plotterp1.trans.y<(abs(tPlotter.tframe.trans.x)-10) THEN
                PlotterZOri:=ACos(Plotterp1.trans.y/abs(tPlotter.tframe.trans.x));
                IF PlotterZOri>PlotA6Max THEN
                    PlotterZOri:=90;
                ENDIF
                Plotterp1.rot:=OrientZYX(-90+PlotterZOri,0,180);
                Plotterp1.trans.y:=Plotterp1.trans.y-((abs(tPlotter.tframe.trans.x)-Ycord1)*(9/((abs(tPlotter.tframe.trans.x)-540))));
            ELSE
                PlotterZOri:=0;
                Plotterp1.rot:=OrientZYX(-90,0,180);
            ENDIF
        ELSE
            RAISE ERR_PLOT_POS;
        ENDIF
        IF PlotterP1.trans.y>(abs(tPlotter.tframe.trans.x)+250) THEN
            Plotterp1.extax:=[(Plotterp1.trans.x+Bed1Wyong.uframe.trans.x),9E+09,9E+09,9E+09,9E+09,9E+09];
        ELSE
            Plotterp1.extax:=[(Plotterp1.trans.x+Bed1Wyong.uframe.trans.x+1000+Abs(tPlotter.tframe.trans.x*Sin(PlotterZOri))),9E+09,9E+09,9E+09,9E+09,9E+09];
        ENDIF


        IF Plotterp2.trans.y>0 THEN
            IF Plotterp2.trans.y<(abs(tPlotter.tframe.trans.x)-10) THEN
                PlotterZOri:=ACos(Plotterp2.trans.y/abs(tPlotter.tframe.trans.x));

                IF PlotterZOri>PlotA6Max THEN
                    PlotterZOri:=90;
                ENDIF
                Plotterp2.rot:=OrientZYX(-90+PlotterZOri,0,180);
                Plotterp2.trans.y:=Plotterp2.trans.y-((abs(tPlotter.tframe.trans.x)-Ycord2)*(9/((abs(tPlotter.tframe.trans.x)-540))));
            ELSE
                PlotterZOri:=0;
                Plotterp2.rot:=OrientZYX(-90,0,180);
            ENDIF
        ELSE
            RAISE ERR_PLOT_POS;
        ENDIF
        IF PlotterP2.trans.y>(abs(tPlotter.tframe.trans.x)+250) THEN
            Plotterp2.extax:=[(Plotterp2.trans.x+Bed1Wyong.uframe.trans.x),9E+09,9E+09,9E+09,9E+09,9E+09];
        ELSE
            Plotterp2.extax:=[(Plotterp2.trans.x+Bed1Wyong.uframe.trans.x+1000+Abs(tPlotter.tframe.trans.x*Sin(PlotterZOri))),9E+09,9E+09,9E+09,9E+09,9E+09];
        ENDIF

        IF Plotterp3.trans.y>0 THEN
            IF Plotterp3.trans.y<(abs(tPlotter.tframe.trans.x)-10) THEN
                PlotterZOri:=ACos(Plotterp3.trans.y/abs(tPlotter.tframe.trans.x));

                IF PlotterZOri>PlotA6Max THEN
                    PlotterZOri:=90;
                ENDIF
                Plotterp3.rot:=OrientZYX(-90+PlotterZOri,0,180);
                Plotterp3.trans.y:=Plotterp3.trans.y-((abs(tPlotter.tframe.trans.x)-Ycord3)*(9/((abs(tPlotter.tframe.trans.x)-540))));

            ELSE
                PlotterZOri:=0;
                Plotterp3.rot:=OrientZYX(-90,0,180);
            ENDIF
        ELSE
            RAISE ERR_PLOT_POS;
        ENDIF
        IF PlotterP3.trans.y>(abs(tPlotter.tframe.trans.x)+250) THEN
            Plotterp3.extax:=[(Plotterp3.trans.x+Bed1Wyong.uframe.trans.x),9E+09,9E+09,9E+09,9E+09,9E+09];
        ELSE
            Plotterp3.extax:=[(Plotterp3.trans.x+Bed1Wyong.uframe.trans.x+1000+Abs(tPlotter.tframe.trans.x*Sin(PlotterZOri))),9E+09,9E+09,9E+09,9E+09,9E+09];
        ENDIF

        IF Plotterp4.trans.y>0 THEN
            IF Plotterp4.trans.y<(abs(tPlotter.tframe.trans.x)-10) THEN
                PlotterZOri:=ACos(Plotterp4.trans.y/abs(tPlotter.tframe.trans.x));
                IF PlotterZOri>PlotA6Max THEN
                    PlotterZOri:=90;
                ENDIF
                Plotterp4.rot:=OrientZYX(-90+PlotterZOri,0,180);
                Plotterp4.trans.y:=Plotterp4.trans.y-((abs(tPlotter.tframe.trans.x)-Ycord4)*(9/((abs(tPlotter.tframe.trans.x)-540))));
            ELSE
                PlotterZOri:=0;
                Plotterp4.rot:=OrientZYX(-90,0,180);
            ENDIF
        ELSE
            RAISE ERR_PLOT_POS;
        ENDIF

        IF PlotterP4.trans.y>(abs(tPlotter.tframe.trans.x)+250) THEN
            Plotterp4.extax:=[(Plotterp4.trans.x+Bed1Wyong.uframe.trans.x),9E+09,9E+09,9E+09,9E+09,9E+09];
        ELSE
            Plotterp4.extax:=[(Plotterp4.trans.x+Bed1Wyong.uframe.trans.x+1000+Abs(tPlotter.tframe.trans.x*Sin(PlotterZOri))),9E+09,9E+09,9E+09,9E+09,9E+09];
        ENDIF

        IF Plotterp1.extax.eax_a>10150 THEN
            Plotterp1.extax.eax_a:=10100;
        ENDIF
        IF Plotterp2.extax.eax_a>10150 THEN
            Plotterp2.extax.eax_a:=10100;
        ENDIF
        IF Plotterp3.extax.eax_a>10150 THEN
            Plotterp3.extax.eax_a:=10100;
        ENDIF
        IF Plotterp4.extax.eax_a>10150 THEN
            Plotterp4.extax.eax_a:=10100;
        ENDIF

        IF Plotterp1.extax.eax_a<0 THEN
            Plotterp1.extax.eax_a:=0;
        ENDIF
        IF Plotterp2.extax.eax_a<0 THEN
            Plotterp2.extax.eax_a:=0;
        ENDIF
        IF Plotterp3.extax.eax_a<0 THEN
            Plotterp3.extax.eax_a:=0;
        ENDIF
        IF Plotterp4.extax.eax_a<0 THEN
            Plotterp4.extax.eax_a:=0;
        ENDIF

        vPlotter:=[100,15,2000,15];

        MoveJ Offs(Plotterp1,0,0,50),v2000,z5,tPlotter\WObj:=Bed1Wyong;
        ConfL\off;
        ConfJ\off;
        MoveL Plotterp1,v10,fine,tPlotter\WObj:=Bed1Wyong;
        WaitTime\inpos,PlotWaitTime;
        MoveL Plotterp2,vPlotter,zPlotter,tPlotter\WObj:=Bed1Wyong;
        WaitTime\inpos,PlotWaitTime;
        MoveL Plotterp3,vPlotter,fine,tPlotter\WObj:=Bed1Wyong;
        WaitTime\inpos,PlotWaitTime;
        MoveL Plotterp4,vPlotter,zPlotter,tPlotter\WObj:=Bed1Wyong;
        WaitTime\inpos,PlotWaitTime;
        MoveL Plotterp1,vPlotter,zPlotter,tPlotter\WObj:=Bed1Wyong;
        MoveL Offs(Plotterp1,0,0,50),v100,z5,tPlotter\WObj:=Bed1Wyong;
        MoveJ Offs(Plotterp1,0,0,200),v500,fine,tPlotter\WObj:=Bed1Wyong;

        ConfL\on;
        ConfJ\on;

    ERROR
        RAISE ;


    ENDPROC

    PROC PlotLineNoLift(num Xcord1,num Ycord1,num Xcord2,num Ycord2)

        IF ToolNum<>4 THEN
            Home;
            Plotter_Pickup;
        ELSE

        ENDIF

        IF Xcord1<=Xcord2 THEN
            Plotterp1.trans:=[-1*Xcord1,Ycord1,PlotterZ];
            Plotterp2.trans:=[-1*Xcord2,Ycord2,PlotterZ];
        ELSE
            Plotterp1.trans:=[-1*Xcord2,Ycord2,PlotterZ];
            Plotterp2.trans:=[-1*Xcord1,Ycord1,PlotterZ];
        ENDIF

        IF Plotterp1.trans.y>0 THEN
            IF ABS(Plotterp1.trans.y)<(abs(tPlotter.tframe.trans.x)-10) THEN
                PlotterZOri:=ACos(Plotterp1.trans.y/abs(tPlotter.tframe.trans.x));
                IF ABS(PlotterZOri)>PlotA6Max THEN
                    PlotterZOri:=90;
                ENDIF
                Plotterp1.rot:=OrientZYX(-90+PlotterZOri,0,180);
                Plotterp1.trans.y:=Plotterp1.trans.y-((abs(tPlotter.tframe.trans.x)-Ycord1)*(9/((abs(tPlotter.tframe.trans.x)-540))));
            ELSEIF Plotterp1.trans.y<2000 THEN
                PlotterZOri:=15;
                Plotterp1.rot:=OrientZYX(-90,0,180);
            ELSE
                PlotterZOri:=0;
                Plotterp1.rot:=OrientZYX(-90,0,180);
            ENDIF
        ELSE
            RAISE ERR_PLOT_POS;
        ENDIF

        IF PlotterP1.trans.y>(abs(tPlotter.tframe.trans.x)+290) THEN
            Plotterp1.extax:=[(Bed1Wyong.uframe.trans.x+Plotterp1.trans.x),9E+09,9E+09,9E+09,9E+09,9E+09];
        ELSE
            Plotterp1.extax:=[(Bed1Wyong.uframe.trans.x+Plotterp1.trans.x+1000+Abs(tPlotter.tframe.trans.x*Sin(PlotterZOri))),9E+09,9E+09,9E+09,9E+09,9E+09];
        ENDIF

        IF Plotterp2.trans.y>0 THEN
            IF Plotterp2.trans.y<(abs(tPlotter.tframe.trans.x)-10) THEN
                PlotterZOri:=ACos(Plotterp2.trans.y/abs(tPlotter.tframe.trans.x));
                IF Plotterp1.trans.y<abs(tPlotter.tframe.trans.x) THEN
                    PlotterZOri:=PlotterZOri+25;
                ENDIF

                IF PlotterZOri>PlotA6Max THEN
                    PlotterZOri:=90;
                ENDIF
                Plotterp2.rot:=OrientZYX(-90+PlotterZOri,0,180);
                Plotterp2.trans.y:=Plotterp2.trans.y-((abs(tPlotter.tframe.trans.x)-Ycord2)*(9/((abs(tPlotter.tframe.trans.x)-540))));
            ELSEIF Plotterp2.trans.y<2000 THEN
                PlotterZOri:=15;
                Plotterp2.rot:=OrientZYX(-90,0,180);
            ELSE
                PlotterZOri:=0;
                Plotterp2.rot:=OrientZYX(-90,0,180);
            ENDIF
        ELSE
            RAISE ERR_PLOT_POS;
        ENDIF

        IF PlotterP2.trans.y>(abs(tPlotter.tframe.trans.x)+250) THEN
            Plotterp2.extax:=[(Plotterp2.trans.x+Bed1Wyong.uframe.trans.x),9E+09,9E+09,9E+09,9E+09,9E+09];
        ELSE
            Plotterp2.extax:=[(Plotterp2.trans.x+Bed1Wyong.uframe.trans.x+1000+Abs(tPlotter.tframe.trans.x*Sin(PlotterZOri))),9E+09,9E+09,9E+09,9E+09,9E+09];
        ENDIF

        IF Plotterp1.extax.eax_a>10150 THEN
            Plotterp1.extax.eax_a:=10100;
        ENDIF
        IF Plotterp2.extax.eax_a>10150 THEN
            Plotterp2.extax.eax_a:=10100;
        ENDIF

        IF Plotterp1.extax.eax_a<0 THEN
            Plotterp1.extax.eax_a:=0;
        ENDIF
        IF Plotterp2.extax.eax_a<0 THEN
            Plotterp2.extax.eax_a:=0;
        ENDIF

        ConfJ\Off;
        ConfL\Off;
        MoveL Plotterp1,v30,zPlotter,tPlotter\WObj:=Bed1Wyong;
        MoveL Plotterp2,vPlotter,fine,tPlotter\WObj:=Bed1Wyong;

        ConfL\on;
        ConfJ\on;

    ERROR
        RAISE ;

    ENDPROC

    PROC PlotLineStartLift(num Xcord1,num Ycord1,num Xcord2,num Ycord2)

        WaitTime\inpos,0.1;
        IF ToolNum<>4 THEN
            Home;
            Plotter_Pickup;
        ENDIF

        IF Xcord1<=Xcord2 THEN
            Plotterp1.trans:=[-1*Xcord1,Ycord1,PlotterZ];
            Plotterp2.trans:=[-1*Xcord2,Ycord2,PlotterZ];
        ELSE
            Plotterp1.trans:=[-1*Xcord2,Ycord2,PlotterZ];
            Plotterp2.trans:=[-1*Xcord1,Ycord1,PlotterZ];
        ENDIF

        IF Plotterp1.trans.y>0 THEN
            IF ABS(Plotterp1.trans.y)<(abs(tPlotter.tframe.trans.x)-10) THEN
                PlotterZOri:=ACos(Plotterp1.trans.y/abs(tPlotter.tframe.trans.x));
                IF ABS(PlotterZOri)>PlotA6Max THEN
                    PlotterZOri:=90;
                ENDIF
                Plotterp1.rot:=OrientZYX(-90+PlotterZOri,0,180);
                Plotterp1.trans.y:=Plotterp1.trans.y-((abs(tPlotter.tframe.trans.x)-Ycord1)*(9/((abs(tPlotter.tframe.trans.x)-540))));
            ELSEIF Plotterp1.trans.y<2000 THEN
                PlotterZOri:=15;
                Plotterp1.rot:=OrientZYX(-90,0,180);
            ELSE
                PlotterZOri:=0;
                Plotterp1.rot:=OrientZYX(-90,0,180);
            ENDIF
        ELSE
            RAISE ERR_PLOT_POS;
        ENDIF

        IF PlotterP1.trans.y>(abs(tPlotter.tframe.trans.x)+290) THEN
            Plotterp1.extax:=[(Bed1Wyong.uframe.trans.x+Plotterp1.trans.x),9E+09,9E+09,9E+09,9E+09,9E+09];
        ELSE
            Plotterp1.extax:=[(Bed1Wyong.uframe.trans.x+Plotterp1.trans.x+1000+Abs(tPlotter.tframe.trans.x*Sin(PlotterZOri))),9E+09,9E+09,9E+09,9E+09,9E+09];
        ENDIF

        IF Plotterp2.trans.y>0 THEN
            IF Plotterp2.trans.y<(abs(tPlotter.tframe.trans.x)-10) THEN
                PlotterZOri:=ACos(Plotterp2.trans.y/abs(tPlotter.tframe.trans.x));
                IF Plotterp1.trans.y<abs(tPlotter.tframe.trans.x) THEN
                    PlotterZOri:=PlotterZOri+25;
                ENDIF

                IF PlotterZOri>PlotA6Max THEN
                    PlotterZOri:=90;
                ENDIF
                Plotterp2.rot:=OrientZYX(-90+PlotterZOri,0,180);
                Plotterp2.trans.y:=Plotterp2.trans.y-((abs(tPlotter.tframe.trans.x)-Ycord2)*(9/((abs(tPlotter.tframe.trans.x)-540))));
            ELSEIF Plotterp2.trans.y<2000 THEN
                PlotterZOri:=15;
                Plotterp2.rot:=OrientZYX(-90,0,180);
            ELSE
                PlotterZOri:=0;
                Plotterp2.rot:=OrientZYX(-90,0,180);
            ENDIF
        ELSE
            RAISE ERR_PLOT_POS;
        ENDIF

        IF PlotterP2.trans.y>(abs(tPlotter.tframe.trans.x)+250) THEN
            Plotterp2.extax:=[(Plotterp2.trans.x+Bed1Wyong.uframe.trans.x),9E+09,9E+09,9E+09,9E+09,9E+09];
        ELSE
            Plotterp2.extax:=[(Plotterp2.trans.x+Bed1Wyong.uframe.trans.x+1000+Abs(tPlotter.tframe.trans.x*Sin(PlotterZOri))),9E+09,9E+09,9E+09,9E+09,9E+09];
        ENDIF

        IF Plotterp1.extax.eax_a>10150 THEN
            Plotterp1.extax.eax_a:=10100;
        ENDIF
        IF Plotterp2.extax.eax_a>10150 THEN
            Plotterp2.extax.eax_a:=10100;
        ENDIF

        IF Plotterp1.extax.eax_a<0 THEN
            Plotterp1.extax.eax_a:=0;
        ENDIF
        IF Plotterp2.extax.eax_a<0 THEN
            Plotterp2.extax.eax_a:=0;
        ENDIF

        ConfJ\Off;
        ConfL\Off;
        MoveJ Offs(Plotterp1,0,0,50),v2000,z5,tPlotter\WObj:=Bed1Wyong;
        ConfL\off;
        ConfJ\off;
        MoveL Plotterp1,v30,zPlotter,tPlotter\WObj:=Bed1Wyong;
        MoveL Plotterp2,vPlotter,fine,tPlotter\WObj:=Bed1Wyong;
        ConfL\on;
        ConfJ\on;

    ERROR
        RAISE ;

    ENDPROC

    PROC PlotLine(num Xcord1,num Ycord1,num Xcord2,num Ycord2)

        WaitTime\inpos,0.1;
        IF ToolNum<>4 THEN
            Home;
            Plotter_Pickup;
        ELSE
            !Check position and move to safe position if needed
            CurrentJoints:=CJointT();
            CurrentPos:=CalcRobT(CurrentJoints,tPlotter\WObj:=Bed1Wyong);

            IF (CurrentPos.trans.z<(Bed1Wyong.uframe.trans.z-30)) OR (((CurrentPos.trans.x+CurrentPos.extax.eax_a)>Bed1Wyong.uframe.trans.x) AND CurrentPos.trans.z<300) THEN
                !Robot in TS
                TPWrite("Jog robot out of tool station AND HOME");
                Stop;
            ENDIF
        ENDIF

        IF Xcord1<=Xcord2 THEN
            Plotterp1.trans:=[-1*Xcord1,Ycord1,PlotterZ];
            Plotterp2.trans:=[-1*Xcord2,Ycord2,PlotterZ];
        ELSE
            Plotterp1.trans:=[-1*Xcord2,Ycord2,PlotterZ];
            Plotterp2.trans:=[-1*Xcord1,Ycord1,PlotterZ];
        ENDIF

        IF Plotterp1.trans.y>0 THEN
            IF ABS(Plotterp1.trans.y)<(abs(tPlotter.tframe.trans.x)-10) THEN
                PlotterZOri:=ACos(Plotterp1.trans.y/abs(tPlotter.tframe.trans.x));
                IF ABS(PlotterZOri)>PlotA6Max THEN
                    PlotterZOri:=90;
                ENDIF
                Plotterp1.rot:=OrientZYX(-90+PlotterZOri,0,180);
                Plotterp1.trans.y:=Plotterp1.trans.y-((abs(tPlotter.tframe.trans.x)-Ycord1)*(9/((abs(tPlotter.tframe.trans.x)-540))));

            ELSEIF Plotterp1.trans.y<2000 THEN
                PlotterZOri:=15;
                Plotterp1.rot:=OrientZYX(-90,0,180);
            ELSE
                PlotterZOri:=0;
                Plotterp1.rot:=OrientZYX(-90,0,180);
            ENDIF
        ELSE
            RAISE ERR_PLOT_POS;
        ENDIF

        IF PlotterP1.trans.y>(abs(tPlotter.tframe.trans.x)+290) THEN
            Plotterp1.extax:=[(Bed1Wyong.uframe.trans.x+Plotterp1.trans.x),9E+09,9E+09,9E+09,9E+09,9E+09];
        ELSE
            Plotterp1.extax:=[(Bed1Wyong.uframe.trans.x+Plotterp1.trans.x+1000+Abs(tPlotter.tframe.trans.x*Sin(PlotterZOri))),9E+09,9E+09,9E+09,9E+09,9E+09];
        ENDIF

        IF Plotterp2.trans.y>0 THEN
            IF Plotterp2.trans.y<(abs(tPlotter.tframe.trans.x)-10) THEN
                PlotterZOri:=ACos(Plotterp2.trans.y/abs(tPlotter.tframe.trans.x));
                IF Plotterp1.trans.y<abs(tPlotter.tframe.trans.x) THEN
                    PlotterZOri:=PlotterZOri+25;
                ENDIF

                IF PlotterZOri>PlotA6Max THEN
                    PlotterZOri:=90;
                ENDIF
                Plotterp2.rot:=OrientZYX(-90+PlotterZOri,0,180);
                Plotterp2.trans.y:=Plotterp2.trans.y-((abs(tPlotter.tframe.trans.x)-Ycord2)*(9/((abs(tPlotter.tframe.trans.x)-540))));

            ELSEIF Plotterp2.trans.y<2000 THEN
                PlotterZOri:=15;
                Plotterp2.rot:=OrientZYX(-90,0,180);
            ELSE
                PlotterZOri:=0;
                Plotterp2.rot:=OrientZYX(-90,0,180);
            ENDIF
        ELSE
            RAISE ERR_PLOT_POS;
        ENDIF

        IF PlotterP2.trans.y>(abs(tPlotter.tframe.trans.x)+250) THEN
            Plotterp2.extax:=[(Plotterp2.trans.x+Bed1Wyong.uframe.trans.x),9E+09,9E+09,9E+09,9E+09,9E+09];
        ELSE
            Plotterp2.extax:=[(Plotterp2.trans.x+Bed1Wyong.uframe.trans.x+1000+Abs(tPlotter.tframe.trans.x*Sin(PlotterZOri))),9E+09,9E+09,9E+09,9E+09,9E+09];
        ENDIF

        IF Plotterp1.extax.eax_a>10150 THEN
            Plotterp1.extax.eax_a:=10100;
        ENDIF
        IF Plotterp2.extax.eax_a>10150 THEN
            Plotterp2.extax.eax_a:=10100;
        ENDIF

        IF Plotterp1.extax.eax_a<0 THEN
            Plotterp1.extax.eax_a:=0;
        ENDIF
        IF Plotterp2.extax.eax_a<0 THEN
            Plotterp2.extax.eax_a:=0;
        ENDIF

        ConfJ\Off;
        ConfL\Off;
        MoveJ Offs(Plotterp1,0,0,50),v2000,z5,tPlotter\WObj:=Bed1Wyong;
        ConfL\off;
        ConfJ\off;
        MoveL Plotterp1,v30,zPlotter,tPlotter\WObj:=Bed1Wyong;
        MoveL Plotterp2,vPlotter,fine,tPlotter\WObj:=Bed1Wyong;
        MoveL Offs(Plotterp2,0,0,50),v100,z5,tPlotter\WObj:=Bed1Wyong;
        MoveJ Offs(Plotterp2,0,0,200),v500,fine,tPlotter\WObj:=Bed1Wyong;

        ConfL\on;
        ConfJ\on;

    ERROR
        RAISE ;

    ENDPROC


    PROC PlotLineEndLift(num Xcord1,num Ycord1,num Xcord2,num Ycord2)

        WaitTime\inpos,0.1;
        IF ToolNum<>4 THEN
            Home;
            Plotter_Pickup;

        ENDIF

        IF Xcord1<=Xcord2 THEN
            Plotterp1.trans:=[-1*Xcord1,Ycord1,PlotterZ];
            Plotterp2.trans:=[-1*Xcord2,Ycord2,PlotterZ];
        ELSE
            Plotterp1.trans:=[-1*Xcord2,Ycord2,PlotterZ];
            Plotterp2.trans:=[-1*Xcord1,Ycord1,PlotterZ];
        ENDIF

        IF Plotterp1.trans.y>0 THEN
            IF ABS(Plotterp1.trans.y)<(abs(tPlotter.tframe.trans.x)-10) THEN
                PlotterZOri:=ACos(Plotterp1.trans.y/abs(tPlotter.tframe.trans.x));
                IF ABS(PlotterZOri)>PlotA6Max THEN
                    PlotterZOri:=90;
                ENDIF
                Plotterp1.rot:=OrientZYX(-90+PlotterZOri,0,180);
                Plotterp1.trans.y:=Plotterp1.trans.y-((abs(tPlotter.tframe.trans.x)-Ycord1)*(9/((abs(tPlotter.tframe.trans.x)-540))));
            ELSEIF Plotterp1.trans.y<2000 THEN
                PlotterZOri:=15;
                Plotterp1.rot:=OrientZYX(-90,0,180);
            ELSE
                PlotterZOri:=0;
                Plotterp1.rot:=OrientZYX(-90,0,180);
            ENDIF
        ELSE
            RAISE ERR_PLOT_POS;
        ENDIF

        IF PlotterP1.trans.y>(abs(tPlotter.tframe.trans.x)+290) THEN
            Plotterp1.extax:=[(Bed1Wyong.uframe.trans.x+Plotterp1.trans.x),9E+09,9E+09,9E+09,9E+09,9E+09];
        ELSE
            Plotterp1.extax:=[(Bed1Wyong.uframe.trans.x+Plotterp1.trans.x+1000+Abs(tPlotter.tframe.trans.x*Sin(PlotterZOri))),9E+09,9E+09,9E+09,9E+09,9E+09];
        ENDIF

        IF Plotterp2.trans.y>0 THEN
            IF Plotterp2.trans.y<(abs(tPlotter.tframe.trans.x)-10) THEN
                PlotterZOri:=ACos(Plotterp2.trans.y/abs(tPlotter.tframe.trans.x));
                IF Plotterp1.trans.y<abs(tPlotter.tframe.trans.x) THEN
                    PlotterZOri:=PlotterZOri+25;
                ENDIF

                IF PlotterZOri>PlotA6Max THEN
                    PlotterZOri:=90;
                ENDIF
                Plotterp2.rot:=OrientZYX(-90+PlotterZOri,0,180);
                Plotterp2.trans.y:=Plotterp2.trans.y-((abs(tPlotter.tframe.trans.x)-Ycord2)*(9/((abs(tPlotter.tframe.trans.x)-540))));

            ELSEIF Plotterp2.trans.y<2000 THEN
                PlotterZOri:=15;
                Plotterp2.rot:=OrientZYX(-90,0,180);
            ELSE
                PlotterZOri:=0;
                Plotterp2.rot:=OrientZYX(-90,0,180);
            ENDIF
        ELSE
            RAISE ERR_PLOT_POS;
        ENDIF

        IF PlotterP2.trans.y>(abs(tPlotter.tframe.trans.x)+250) THEN
            Plotterp2.extax:=[(Plotterp2.trans.x+Bed1Wyong.uframe.trans.x),9E+09,9E+09,9E+09,9E+09,9E+09];
        ELSE
            Plotterp2.extax:=[(Plotterp2.trans.x+Bed1Wyong.uframe.trans.x+1000+Abs(tPlotter.tframe.trans.x*Sin(PlotterZOri))),9E+09,9E+09,9E+09,9E+09,9E+09];
        ENDIF

        IF Plotterp1.extax.eax_a>10150 THEN
            Plotterp1.extax.eax_a:=10100;
        ENDIF
        IF Plotterp2.extax.eax_a>10150 THEN
            Plotterp2.extax.eax_a:=10100;
        ENDIF

        IF Plotterp1.extax.eax_a<0 THEN
            Plotterp1.extax.eax_a:=0;
        ENDIF
        IF Plotterp2.extax.eax_a<0 THEN
            Plotterp2.extax.eax_a:=0;
        ENDIF

        ConfJ\Off;
        ConfL\Off;
        MoveL Plotterp1,v30,zPlotter,tPlotter\WObj:=Bed1Wyong;
        MoveL Plotterp2,vPlotter,fine,tPlotter\WObj:=Bed1Wyong;
        MoveL Offs(Plotterp2,0,0,50),v100,z5,tPlotter\WObj:=Bed1Wyong;
        MoveJ Offs(Plotterp2,0,0,200),v500,fine,tPlotter\WObj:=Bed1Wyong;

        ConfL\on;
        ConfJ\on;

    ERROR
        RAISE ;

    ENDPROC

    PROC PlotArc(num StartXcord,num StartYcord,num MidXcord,num MidYcord,num EndXcord,num EndYcord)
        IF ToolNum<>4 THEN
            Home;
            Plotter_Pickup;
        ELSE
            !Check position and move to safe position if needed
            !Check position and move to safe position if needed
            CurrentJoints:=CJointT();
            CurrentPos:=CalcRobT(CurrentJoints,tPlotter\WObj:=Bed1Wyong);

            IF (CurrentPos.trans.z<(Bed1Wyong.uframe.trans.z-30)) OR (((CurrentPos.trans.x+CurrentPos.extax.eax_a)>Bed1Wyong.uframe.trans.x) AND CurrentPos.trans.z<300) THEN
                !Robot in TS
                TPWrite("Jog robot out of tool station AND HOME");
                Stop;
            ENDIF
        ENDIF

        !Plot Circle
        Plotterc5.trans:=[(-1*StartXcord),StartYcord,PlotterZ];
        PlotterTemp.trans:=[Plotterc5.trans.x,Plotterc5.trans.y,PlotterZ];

        IF PlotterTemp.trans.y>0 THEN
            IF PlotterTemp.trans.y<(abs(tPlotter.tframe.trans.x)-10) THEN
                PlotterZOri:=ACos(PlotterTemp.trans.y/abs(tPlotter.tframe.trans.x));
                IF PlotterZOri>PlotA6Max THEN
                    PlotterZOri:=90;
                ENDIF
                PlotterTemp.rot:=OrientZYX(-90+PlotterZOri,0,180);
                PlotterTemp.trans.y:=PlotterTemp.trans.y-((abs(tPlotter.tframe.trans.x)-StartYcord)*(9/((abs(tPlotter.tframe.trans.x)-540))));
            ELSE
                PlotterTemp.rot:=OrientZYX(-90,0,180);
            ENDIF
        ELSE
            RAISE ERR_PLOT_POS;
        ENDIF

        IF PlotterTemp.trans.y+Bed1.uframe.trans.y>2800 THEN
            PlotterTemp.extax.eax_a:=(PlotterTemp.trans.x+Bed1Wyong.uframe.trans.x);
        ELSE
            PlotterTemp.extax.eax_a:=(PlotterTemp.trans.x+Bed1Wyong.uframe.trans.x+1000+Abs(tPlotter.tframe.trans.x*Sin(PlotterZOri)));
        ENDIF

        IF PlotterTemp.extax.eax_a>10150 THEN
            PlotterTemp.extax.eax_a:=10100;
        ELSEIF PlotterTemp.extax.eax_a<0 THEN
            PlotterTemp.extax.eax_a:=0;
        ENDIF

        WaitTime\inpos,0.1;
        ConfJ\Off;
        ConfL\Off;

        MoveJ Offs(PlotterTemp,0,0,50),v1500,z5,tPlotter\WObj:=Bed1Wyong;
        MoveL PlotterTemp,v10,fine,tPlotter\WObj:=Bed1Wyong;

        PlotterTemp2.trans:=[(-1*MidXcord),MidYcord,PlotterZ];
        IF PlotterTemp2.trans.y>0 THEN
            IF PlotterTemp2.trans.y<(abs(tPlotter.tframe.trans.x)-10) THEN
                PlotterZOri:=ACos(PlotterTemp2.trans.y/abs(tPlotter.tframe.trans.x));
                IF PlotterZOri>PlotA6Max THEN
                    PlotterZOri:=90;
                ENDIF
                PlotterTemp2.rot:=OrientZYX(-90+PlotterZOri,0,180);
                PlotterTemp2.trans.y:=PlotterTemp2.trans.y-((abs(tPlotter.tframe.trans.x)-MidYcord)*(9/((abs(tPlotter.tframe.trans.x)-540))));
            ELSE
                PlotterZOri:=0;
                PlotterTemp3.rot:=OrientZYX(-90,0,180);
            ENDIF
        ELSE
            RAISE ERR_PLOT_POS;
        ENDIF
        IF PlotterTemp2.trans.y+Bed1.uframe.trans.y>2800 THEN
            PlotterTemp2.extax.eax_a:=(PlotterTemp2.trans.x+Bed1Wyong.uframe.trans.x);
        ELSE
            PlotterTemp2.extax.eax_a:=(PlotterTemp2.trans.x+Bed1Wyong.uframe.trans.x+1000+Abs(tPlotter.tframe.trans.x*Sin(PlotterZOri)));
        ENDIF

        IF PlotterTemp2.extax.eax_a>10150 THEN
            PlotterTemp2.extax.eax_a:=10100;
        ELSEIF PlotterTemp2.extax.eax_a<0 THEN
            PlotterTemp2.extax.eax_a:=0;
        ENDIF

        PlotterTemp3.trans:=[(-1*EndXcord),EndYcord,PlotterZ];
        IF PlotterTemp3.trans.y>0 THEN
            IF PlotterTemp3.trans.y<(abs(tPlotter.tframe.trans.x)-10) THEN
                PlotterZOri:=ACos(PlotterTemp3.trans.y/abs(tPlotter.tframe.trans.x));
                IF PlotterZOri>PlotA6Max THEN
                    PlotterZOri:=90;
                ENDIF
                PlotterTemp3.rot:=OrientZYX(-90+PlotterZOri,0,180);
                PlotterTemp3.trans.y:=PlotterTemp3.trans.y-((abs(tPlotter.tframe.trans.x)-EndYcord)*(9/((abs(tPlotter.tframe.trans.x)-540))));
            ELSE
                PlotterZOri:=0;
                PlotterTemp3.rot:=OrientZYX(-90,0,180);
            ENDIF
        ELSE
            RAISE ERR_PLOT_POS;
        ENDIF
        IF PlotterTemp3.trans.y+Bed1Wyong.uframe.trans.y>2800 THEN
            PlotterTemp3.extax:=[(PlotterTemp3.trans.x+Bed1Wyong.uframe.trans.x),9E+09,9E+09,9E+09,9E+09,9E+09];
        ELSE
            PlotterTemp3.extax:=[(PlotterTemp3.trans.x+Bed1Wyong.uframe.trans.x+1000+Abs(tPlotter.tframe.trans.x*Sin(PlotterZOri))),9E+09,9E+09,9E+09,9E+09,9E+09];
        ENDIF

